(* PLC project Система умного дома.project, CODESYS CODESYS V3.5 SP17 Patch 3 *)
(* stored: creationDateTime 2026-04-06T20:38:17.5908527, modificationDateTime 2026-03-25T09:46:39.3897592 *)

TYPE E_ALERT_PRIORITY : (ALERT_PRIORITY_NONE := 0, ALERT_PRIORITY_LOW := 1, ALERT_PRIORITY_MEDIUM := 2, ALERT_PRIORITY_HIGH := 3, ALERT_PRIORITY_CRITICAL := 4) USINT;
END_TYPE

TYPE E_Behavior_Mode : (BEHAVIOR_HOME := 0, BEHAVIOR_AWAY := 1, BEHAVIOR_NIGHT := 2, BEHAVIOR_MAINTENANCE := 3) INT;
END_TYPE

TYPE E_Gateway_Command_Type : (CMD_NONE := 0, CMD_SET_SCENARIO := 1, CMD_SET_LIGHT := 2, CMD_SET_SOCKET := 3, CMD_SET_SECURITY := 4, CMD_SET_TEMP := 5, CMD_SET_VENT := 6, CMD_SET_BLINDS := 7, CMD_TELEGRAM_MSG := 8, CMD_SYNC_TIME := 9, CMD_RESET_ERRORS := 10, CMD_SET_CONFIG := 11) USINT;
END_TYPE

TYPE E_Lifetime_Device_Type : (LIFETIME_DEVICE_PUMP := 1, LIFETIME_DEVICE_FAN := 2) USINT;
END_TYPE

TYPE E_Outdoor_Mode : (OUTDOOR_MODE_AUTO := 0, OUTDOOR_MODE_PARTY := 1, OUTDOOR_MODE_SECURITY := 2, OUTDOOR_MODE_ECONOMY := 3, OUTDOOR_MODE_MANUAL := 4) USINT;
END_TYPE

TYPE E_PLC_ROLE : (ROLE_UNDEFINED := 0, ROLE_ACTIVE := 1, ROLE_STANDBY := 2, ROLE_OFFLINE := 3) USINT;
END_TYPE

TYPE E_Rule_Action_Type : (ACTION_NONE := 0, ACTION_SET_FLOOR_HEATING := 1, ACTION_SET_LIGHTING_BASE := 2, ACTION_SET_LIGHTING_ACCENT := 3, ACTION_SET_SOCKET := 4, ACTION_SET_VENTILATION := 5, ACTION_SET_BLINDS := 6, ACTION_ACTIVATE_SCENARIO := 7, ACTION_TOGGLE_LIGHTING := 8, ACTION_TOGGLE_SOCKET := 9) USINT;
END_TYPE

TYPE E_Rule_Comparison : (COMP_NONE := 0, COMP_EQ := 1, COMP_GT := 2, COMP_LT := 3, COMP_GE := 4, COMP_LE := 5, COMP_IN_RANGE := 6, COMP_TRUE := 7, COMP_FALSE := 8) USINT;
END_TYPE

TYPE E_Rule_Condition_Type : (COND_NONE := 0, COND_AIR_TEMP := 1, COND_FLOOR_TEMP := 2, COND_HUMIDITY := 3, COND_CO2 := 4, COND_METHANE := 5, COND_CO := 6, COND_DOOR_WINDOW := 7, COND_FLOOD := 8, COND_SMOKE := 9, COND_MOTION := 10, COND_TIME_OF_DAY := 11, COND_DAY_OF_WEEK := 12) USINT;
END_TYPE

TYPE E_SCENARIO_SOURCE : (SRC_NONE := 0, SRC_OPERATOR := 1, SRC_GATEWAY := 2, SRC_RULE := 3, SRC_SAFETY := 4, SRC_POLICY := 5) INT;
END_TYPE

TYPE E_SCENARIO_TYPE : (SCENARIO_NONE := 0, SCENARIO_MORNING := 1, SCENARIO_EVENING := 2, SCENARIO_AWAY := 3, SCENARIO_PARTY := 4, SCENARIO_SLEEP := 5, SCENARIO_EMERGENCY := 6, SCENARIO_PRESENCE := 7) USINT;
END_TYPE

TYPE E_SENSOR_TYPE : (SENSOR_TYPE_NONE := 0, SENSOR_TYPE_DOOR_WINDOW := 5, SENSOR_TYPE_GLASS_BREAK := 6, SENSOR_TYPE_FLOOD := 7, SENSOR_TYPE_SMOKE := 8, SENSOR_TYPE_GAS_METHANE := 1, SENSOR_TYPE_GAS_CO := 2, SENSOR_TYPE_TEMP_FLOOR := 3, SENSOR_TYPE_TEMP_AIR := 4, SENSOR_TYPE_CO2 := 9) USINT;
END_TYPE

TYPE E_System_Operating_Mode : (MODE_NORMAL := 0, MODE_DEGRADED := 1, MODE_SAFE_STOP := 2, MODE_FREEZE_PROTECTION := 3) INT;
END_TYPE

TYPE E_System_Root_Cause : (ROOT_NONE := 0, ROOT_FIRE := 1, ROOT_GAS_LEAK := 2, ROOT_CO_WARNING := 3, ROOT_CO_CRITICAL := 4, ROOT_WATER_LEAK := 5, ROOT_IO_OFFLINE := 6, ROOT_COMM_FAULT := 7, ROOT_SENSOR_FAULT := 8, ROOT_SUBSYSTEM_FAULT := 9, ROOT_WATCHDOG_FAULT := 10) INT;
END_TYPE

TYPE E_System_Severity : (SEV_NORMAL := 0, SEV_WARNING := 1, SEV_DEGRADED := 2, SEV_CRITICAL := 3) INT;
END_TYPE

TYPE E_Trend_Parameter_Type : (TREND_PARAM_NONE := 0, TREND_PARAM_TEMP_AIR := 1, TREND_PARAM_TEMP_FLOOR := 2, TREND_PARAM_PRESSURE := 3, TREND_PARAM_PUMP_CURRENT := 4, TREND_PARAM_GAS_METHANE := 5, TREND_PARAM_GAS_CO := 6) USINT;
END_TYPE

TYPE E_TwoFactor_Method : (TF_METHOD_NONE := 0, TF_METHOD_RFID := 1, TF_METHOD_TOTP := 2, TF_METHOD_BOTH := 3) USINT;
END_TYPE

TYPE E_VALVE_TYPE : (VALVE_NC := 1, VALVE_NO := 2) USINT;
END_TYPE

TYPE E_VENTILATION_LOCATION : (VENT_LOCATION_NONE := 0, VENT_LOCATION_BASEMENT_GAME_ROOM := 1, VENT_LOCATION_BASEMENT_GYM := 2, VENT_LOCATION_BASEMENT_BOILER_ROOM := 3, VENT_LOCATION_BATHROOM_1F := 4, VENT_LOCATION_BATHROOM_2F := 5, VENT_LOCATION_MASTER_BATHROOM := 6, VENT_LOCATION_LAUNDRY := 7, VENT_LOCATION_KITCHEN := 8) USINT;
END_TYPE

TYPE E_VENTILATION_UNIT_TYPE : (VENTILATION_TYPE_NONE := 0, VENTILATION_TYPE_SUPPLY := 1, VENTILATION_TYPE_EXHAUST := 2) USINT;
END_TYPE

TYPE E_Valve_Test_Result : (TEST_RESULT_NONE := 0, TEST_RESULT_PASSED := 1, TEST_RESULT_CURRENT_DEVIATION := 2, TEST_RESULT_TIME_DEVIATION := 3, TEST_RESULT_STALL := 4, TEST_RESULT_LIMIT_SWITCH_FAIL := 5, TEST_RESULT_ABORTED := 6) USINT;
END_TYPE

TYPE E_WEATHER_COMPENSATION_METHOD : (WEATHER_COMP_NONE := 0, WEATHER_COMP_OUTDOOR_RESET := 1) USINT;
END_TYPE

TYPE E_Zone_Access_Level : (ZONE_ACCESS_NONE := 0, ZONE_ACCESS_VIEW := 1, ZONE_ACCESS_CONTROL := 2, ZONE_ACCESS_CONFIG := 3, ZONE_ACCESS_FULL := 4) USINT;
END_TYPE

TYPE ST_Alarm_Record : STRUCT
  ID : UDINT;
  Timestamp_MS : UDINT;
  Source : STRING(20);
  Source_ID : BYTE;
  Message : STRING(100);
  Severity : E_ALERT_PRIORITY;
  Is_Active : BOOL;
  Is_Acknowledged : BOOL;
END_STRUCT;
END_TYPE

TYPE ST_Astro_Time : STRUCT
  sunrise_ms : UDINT := 0;
  sunset_ms : UDINT := 0;
  is_daylight : BOOL := FALSE;
END_STRUCT;
END_TYPE

TYPE ST_BlackBox_Record : STRUCT
  Timestamp : UDINT;
  Gas_Methane_LEL : REAL;
  Gas_CO_PPM : REAL;
  Flood_Active : BOOL;
  Fire_Active : BOOL;
  Valve_Gas_Status : BYTE;
  Valve_Water_Status : BYTE;
  PLC_Active_ID : BYTE;
  System_Mode : BYTE;
  First_Fault_Type : BYTE;
  First_Fault_Source : BYTE;
  First_Fault_Active : BOOL;
  System_Severity : BYTE;
  Root_Cause : BYTE;
  Watchdog_Fault : BOOL;
END_STRUCT;
END_TYPE

TYPE ST_Boiler_Status : STRUCT
  Active : BOOL;
  Running : BOOL;
  Warning : BOOL;
  Error : BOOL;
  Error_ID : WORD;
  Power_Percent : REAL;
  Current_Power : REAL;
  Work_Seconds : UDINT;
  Work_Hours : REAL;
  Resource_Percent : REAL := 100.0;
  Last_Start : DT;
END_STRUCT;
END_TYPE

TYPE ST_Calibration_Family_Summary : STRUCT
  active : BOOL;
  status : INT;
  sensor_count : INT;
  verification_active_count : INT;
  failed_count : INT;
  max_deviation_percent : REAL;
  summary_text : STRING(160);
END_STRUCT;
END_TYPE

TYPE ST_Calibration_Sensor_Summary : STRUCT
  active : BOOL;
  status : INT;
  calibrated_value : REAL;
  deviation_percent : REAL;
  verification_active : BOOL;
  verification_failed : BOOL;
  record_index : INT;
  label : STRING(64);
  summary_text : STRING(160);
END_STRUCT;
END_TYPE

TYPE ST_Component_Maintenance : STRUCT
  Is_Faulty : BOOL;
  Is_In_Maintenance : BOOL;
  Fallback_Value : REAL;
  Use_Last_Good_Value : BOOL;
END_STRUCT;
END_TYPE

TYPE ST_DHW_Config : STRUCT
  Target_Temp : REAL := 55.0;
  Hysteresis : REAL := 2.0;
  Circulation_Schedule_Enabled : BOOL := TRUE;
  Circulation_Start : TOD := TOD#06:00;
  Circulation_End : TOD := TOD#23:00;
  Night_Mode_Enabled : BOOL := TRUE;
  Anti_Legionella_Enabled : BOOL := TRUE;
  Anti_Legionella_Day : UINT := 7;
  Degraded_Target_Delta : REAL := 5.0;
END_STRUCT;
END_TYPE

TYPE ST_DHW_Status : STRUCT
  Temp : REAL;
  Pressure : REAL;
  Heating_Pump_On : BOOL;
  Circ_Pump_On : BOOL;
  Warning : BOOL;
  Error : BOOL;
  Error_ID : WORD;
END_STRUCT;
END_TYPE

TYPE ST_Device_Health : STRUCT
  Health_Score : BYTE := 100;
  Total_Runtime_Hours : UDINT;
  Starts_Count : UDINT;
  Last_Start_Current : REAL;
  Avg_Start_Current : REAL;
  Sample_Count : UDINT;
  Current_Sum : REAL;
  Maintenance_Required : BOOL;
  Warning_Message : STRING(50);
END_STRUCT;
END_TYPE

TYPE ST_Diagnostic_Event : STRUCT
  Code : UDINT;
  Severity : INT;
  Active : BOOL;
  Timestamp : UDINT;
  Source : INT;
END_STRUCT;
END_TYPE

TYPE ST_EVENT : STRUCT
  Event_ID : UDINT;
  Event_Type : UINT;
  Timestamp : UDINT;
  Param1 : UDINT;
  Param2 : UDINT;
END_STRUCT;
END_TYPE

TYPE ST_Flood_Config : STRUCT
  Emergency_Two_Stage_Enabled : BOOL := TRUE;
  Valve_Test_Period_Days : UINT := 7;
  Current_Threshold_MA : REAL := 500.0;
  sensor_to_valve_map : ARRAY[1..GVL_CONSTANTS.C_MAX_FLOOD_SENSORS] OF INT := [1, 1, 1, 1, 2, 2, 2, 2, 3, 3, 3, 3];
END_STRUCT;
END_TYPE

TYPE ST_Flood_Global_Config : STRUCT
  valve_types : ARRAY[1..GVL_CONSTANTS.C_MAX_FLOOD_VALVES] OF E_VALVE_TYPE := [GVL_CONSTANTS.C_MAX_FLOOD_VALVES(E_VALVE_TYPE.VALVE_NC)];
  sensor_to_valve_map : ARRAY[1..GVL_CONSTANTS.C_MAX_FLOOD_SENSORS] OF BYTE := [1, 1, 1, 2, 2, 2, 2, 0, 0, 0];
  min_duration_ms : UDINT := 5000;
  warning_duration_ms : UDINT := 30000;
END_STRUCT;
END_TYPE

TYPE ST_FloorHeating_Circuit_Config : STRUCT
  circuit_id : BYTE := 0;
  zone : BYTE := 0;
  manifold_id : BYTE := 1;
  sensor_id : BYTE := 1;
  valve_id : BYTE := 1;
  control_type : BYTE := 1;
  design_temp : REAL := 35.0;
  min_temp : REAL := 20.0;
  max_temp : REAL := 45.0;
  pid_kp : REAL := 2.0;
  pwm_period_s : UINT := 600;
END_STRUCT;
END_TYPE

TYPE ST_FloorHeating_Global_Config : STRUCT
  enable_floor_heating : BOOL := TRUE;
  anti_freeze_temp : REAL := 7.0;
  overheat_temp : REAL := 45.0;
  weather_compensation_enabled : BOOL := TRUE;
  total_circuits : BYTE := 16;
END_STRUCT;
END_TYPE

TYPE ST_FloorHeating_Manifold_Config : STRUCT
  manifold_id : BYTE;
  location : STRING(30);
  nominal_flow : REAL;
  enable_pump : BOOL;
  circuits : ARRAY[1..GVL_CONSTANTS.C_MAX_CIRCUITS_PER_MANIFOLD] OF ST_FloorHeating_Circuit_Config;
END_STRUCT;
END_TYPE

TYPE ST_Gas_Valve_Configuration : STRUCT
  valve_id : BYTE := 0;
  valve_type : E_VALVE_TYPE := E_VALVE_TYPE.VALVE_NC;
  close_time_seconds : UDINT := 10;
  open_time_seconds : UDINT := 10;
  emergency_open_allowed : BOOL := FALSE;
END_STRUCT;
END_TYPE

TYPE ST_Gateway_Command : STRUCT
  command_id : UDINT;
  timestamp_ms : UDINT;
  operator_id : STRING(10);
  command_type : E_Gateway_Command_Type;
  target_zone : BYTE;
  target_value : REAL;
  target_on_off : BOOL;
  target_scenario : E_SCENARIO_TYPE;
  target_armed : BOOL;
  target_pin : STRING(4);
  target_2fa_code : STRING(6);
  telegram_msg : STRING(200);
  source_ip : STRING(15);
  crc32 : DWORD;
END_STRUCT;
END_TYPE

TYPE ST_Heating_Config : STRUCT
  Weather_Comp_Enabled : BOOL := TRUE;
  Weather_Coef : REAL := 0.1;
  Freeze_Threshold : REAL := 7.0;
  Overheat_Threshold : REAL := 45.0;
  Night_Reduction : REAL := 3.0;
  Target_Floor_Temp : REAL := 28.0;
  Target_Room_Temp : REAL := 22.0;
  Hysteresis : REAL := 0.5;
END_STRUCT;
END_TYPE

TYPE ST_History_Record : STRUCT
  timestamp_ms : UDINT := 0;
  event_code : WORD := 0;
  event_value : REAL := 0.0;
  unit : BYTE := 0;
  zone_id : BYTE := 0;
  operator_id : STRING(10) := '';
  priority : E_ALERT_PRIORITY := E_ALERT_PRIORITY.ALERT_PRIORITY_NONE;
END_STRUCT;
END_TYPE

TYPE ST_Lifetime_Status : STRUCT
  device_id : BYTE;
  runtime_hours : UDINT;
  start_count : UDINT;
  remaining_hours : UDINT;
  remaining_percent : BYTE;
  maintenance_required : BOOL;
  last_calc_timestamp : UDINT;
END_STRUCT;
END_TYPE

TYPE ST_Maintenance_Access_Config : STRUCT
  maintenance_enabled : BOOL := FALSE;
  max_duration_minutes : UDINT := 60;
  requires_two_person : BOOL := TRUE;
  access_level_required : BYTE := 2;
END_STRUCT;
END_TYPE

TYPE ST_Manifold_Status : STRUCT
  Pump_On : BOOL;
  Pump_Current : REAL;
  Pressure : REAL;
  Temp_Supply : REAL;
  Temp_Return : REAL;
  Valve_Pos : REAL;
  Error : BOOL;
  Error_ID : WORD;
  Health : ST_Device_Health;
END_STRUCT;
END_TYPE

TYPE ST_Operator_Zone_Rights : STRUCT
  operator_id : STRING(10);
  global_access_level : BYTE := 0;
  zone_masks : DWORD;
  last_modified : UDINT;
END_STRUCT;
END_TYPE

TYPE ST_Outdoor_Zone_Config : STRUCT
  zone_id : BYTE := 0;
  lighting_circuit_id : BYTE := 0;
  auto_enabled : BOOL := TRUE;
  party_mode_enabled : BOOL := FALSE;
END_STRUCT;
END_TYPE

TYPE ST_Owen_Analog_Value : STRUCT
  rValue : REAL;
  uiCycleTime : UINT;
  wStatus : WORD;
END_STRUCT;
END_TYPE

TYPE ST_Persist : STRUCT
  System_Mode : E_System_Operating_Mode;
  Safety_Gas_Latched : BOOL;
  Safety_Smoke_Latched : BOOL;
  Safety_Leak_Latched : BOOL;
  DHW_Heating_Pump : BOOL;
  Valid : BOOL;
  Version : UINT := 1;
END_STRUCT;
END_TYPE

TYPE ST_Rule : STRUCT
  Action_Type : INT;
  Action_Target_ID : INT;
  Action_Value : REAL;
  Condition_Type : INT;
  Condition_Target_ID : INT;
  Condition_Op : INT;
  Condition_Value : REAL;
  Condition_Value_Max : REAL;
END_STRUCT;
END_TYPE

TYPE ST_Rule_Action : STRUCT
  Active : BOOL;
  Triggered : BOOL;
  Action_Type : E_Rule_Action_Type;
  Target_ID : BYTE;
  Value : REAL;
END_STRUCT;
END_TYPE

TYPE ST_Scenario_Config : STRUCT
  scenario_id : E_SCENARIO_TYPE;
  lighting_level_base : BYTE := 100;
  lighting_level_accent : BYTE := 100;
  floor_heating_adjust_celsius : REAL := 0.0;
  ventilation_speed_percent : BYTE := 50;
  sockets_enabled : BOOL := TRUE;
  blinds_position_percent : BYTE := 0;
  Presence_Simulation_Enabled : BOOL := FALSE;
END_STRUCT;
END_TYPE

TYPE ST_Scenario_Transition_Config : STRUCT
  current_scenario : E_SCENARIO_TYPE;
  target_scenario : E_SCENARIO_TYPE;
  min_duration_minutes : UDINT := 5;
  transition_allowed : BOOL := FALSE;
END_STRUCT;
END_TYPE

TYPE ST_Security_Global_Config : STRUCT
  PIN_Code : STRING(4) := '1234';
  Phones : ARRAY[1..GVL_CONSTANTS.C_MAX_SECURITY_PHONES] OF STRING(15);
  entry_delay_seconds : UDINT := 30;
  exit_delay_seconds : UDINT := 60;
  alarm_duration_seconds : UDINT := 180;
  two_person_timeout_seconds : UDINT := 120;
  max_access_attempts : BYTE := 3;
  auto_arm_enabled : BOOL := FALSE;
  auto_arm_time_ms : UDINT := 0;
  enable_2fa : BOOL := TRUE;
  gate_open_pulse_ms : UDINT := GVL_CONSTANTS.C_MS_IN_SECOND;
  wicket_open_pulse_ms : UDINT := GVL_CONSTANTS.C_MS_IN_SECOND;
  lock_open_pulse_ms : UDINT := GVL_CONSTANTS.C_MS_IN_SECOND;
  lock_close_pulse_ms : UDINT := GVL_CONSTANTS.C_MS_IN_SECOND;
  bypass_motion : ARRAY[1..16] OF BOOL;
  bypass_doors : ARRAY[1..GVL_CONSTANTS.C_MAX_DOOR_SENSORS] OF BOOL;
  bypass_windows : ARRAY[1..16] OF BOOL;
END_STRUCT;
END_TYPE

TYPE ST_Security_Zone_State : STRUCT
  Armed : BOOL;
  Alarm : BOOL;
  Bypassed : BOOL;
  Last_Trigger_Time : DT;
  Trigger_Count : UINT;
END_STRUCT;
END_TYPE

TYPE ST_Sensor_Calibration_Record : STRUCT
  sensor_id : UDINT := 0;
  sensor_type : E_SENSOR_TYPE;
  zone_id : BYTE := 0;
  offset : REAL := 0.0;
  multiplier : REAL := 1.0;
  last_calibration_timestamp : UDINT := 0;
  verification_passed : BOOL := FALSE;
END_STRUCT;
END_TYPE

TYPE ST_State_Snapshot : STRUCT
  timestamp_ms : UDINT := 0;
  operator_id : STRING(10) := '';
  scenario_id : E_SCENARIO_TYPE := E_SCENARIO_TYPE.SCENARIO_NONE;
  lighting_levels : ARRAY[1..GVL_CONSTANTS.C_MAX_LIGHTING_ZONES] OF BYTE;
  floor_heating_setpoints : ARRAY[1..GVL_CONSTANTS.C_MAX_HEATING_CIRCUITS] OF REAL;
  alarm_active : BOOL := FALSE;
  crc32 : DWORD := 0;
END_STRUCT;
END_TYPE

TYPE ST_System_Diagnostics : STRUCT
  Freeze_Hardware_Event_Pending : BOOL;
  Freeze_Hardware_Event_Text : STRING(200);
  Backup_Pump_Fault : BOOL;
  Electric_Heater_Fault : BOOL;
  Backup_Pump_Recovered_After_Retry : BOOL;
  Electric_Heater_Recovered_After_Retry : BOOL;
  Backup_Pump_Out_Of_Service : BOOL;
  Electric_Heater_Out_Of_Service : BOOL;
  Pump_Exercise_Active : BOOL;
  Pump_Exercise_Failed : BOOL;
  Pump_Exercise_Last_Equipment : STRING(80);
  Pump_Exercise_Last_Result : STRING(120);
  Pump_Exercise_No_Feedback_Count : INT;
  Manifold_Pump_Exercise_Count : ARRAY[1..GVL_CONSTANTS.C_MAX_MANIFOLDS] OF UDINT;
  DHW_Heating_Pump_Exercise_Count : UDINT;
  DHW_Circ_Pump_Exercise_Count : UDINT;
  Backup_Pump_Exercise_Count : UDINT;
  Pump_Exercise_Event_Seq : UDINT;
  Pump_Exercise_Journal_1 : STRING(200);
  Pump_Exercise_Journal_2 : STRING(200);
  Pump_Exercise_Journal_3 : STRING(200);
  Pump_Exercise_Journal_Last_Seq : UDINT;
  Pump_Maintenance_Required : BOOL;
  Pump_Maintenance_Warning : BOOL;
  Manifold_Pump_Out_Of_Service : ARRAY[1..GVL_CONSTANTS.C_MAX_MANIFOLDS] OF BOOL;
  DHW_Heating_Pump_Out_Of_Service : BOOL;
  DHW_Circ_Pump_Out_Of_Service : BOOL;
  Maintenance_Last_Action : STRING(120);
  Operator_Action_Blocked : BOOL;
  Operator_Block_Reason : STRING(160);
  Operator_Last_Forbidden_Action : STRING(160);
  Operator_Journal_1 : STRING(200);
  Operator_Journal_2 : STRING(200);
  Operator_Journal_3 : STRING(200);
  Operator_Journal_Event_Seq : UDINT;
  Operator_Journal_Last_Seq : UDINT;
  Dangerous_Action_Pending_Confirm : BOOL;
  Dangerous_Action_Confirm_Text : STRING(160);
  Dangerous_Action_Confirm_Deadline_MS : UDINT;
  User_Access_Level_Active : INT;
  User_Access_Denied : BOOL;
  User_Access_Deny_Reason : STRING(160);
  Valve_Test_Mode_Active : BOOL;
  Valve_Test_Deadline_MS : UDINT;
  Valve_Test_Remaining_MS : UDINT;
  Valve_Test_Validation_OK : BOOL;
  Valve_Test_Validation_Text : STRING(160);
  Valve_Test_Forced_Close : BOOL;
  Water_Valve_Test_Mode_Active : BOOL;
  Water_Valve_Test_Deadline_MS : UDINT;
  Water_Valve_Test_Remaining_MS : UDINT;
  Water_Valve_Test_Validation_OK : BOOL;
  Water_Valve_Test_Validation_Text : STRING(160);
  Water_Valve_Test_Forced_Close : BOOL;
  Gas_Valve_Test_Mode_Active : BOOL;
  Gas_Valve_Test_Deadline_MS : UDINT;
  Gas_Valve_Test_Remaining_MS : UDINT;
  Gas_Valve_Test_Validation_OK : BOOL;
  Gas_Valve_Test_Validation_Text : STRING(160);
  Gas_Valve_Test_Forced_Close : BOOL;
  Active_Leak_Sensor_Index : INT;
  Active_Gas_Sensor_Index : INT;
  Active_Leak_Zone_Name : STRING(80);
  Active_Gas_Zone_Name : STRING(80);
  Water_Valve_Test_Context : STRING(160);
  Gas_Valve_Test_Context : STRING(160);
  Water_Recovery_Target_Zone_Index : INT;
  Gas_Recovery_Target_Zone_Index : INT;
  Water_Recovery_Selective_Allowed : BOOL;
  Gas_Recovery_Selective_Allowed : BOOL;
  Water_Recovery_Selective_Text : STRING(160);
  Gas_Recovery_Selective_Text : STRING(160);
  Water_Recovery_Physical_Active : BOOL;
  Water_Recovery_Physical_Zone_Name : STRING(80);
  Water_Zone_Open_Fault : ARRAY[1..32] OF BOOL;
  Water_Zone_Close_Fault : ARRAY[1..32] OF BOOL;
  Water_Valve_Exercise_Last_Zone : INT;
  Water_Valve_Exercise_Last_Result : STRING(160);
  Water_Zone_Critical_Close_Fault : ARRAY[1..32] OF BOOL;
  Water_Close_Fault_Active : BOOL;
  Water_Close_Fault_Zone_Name : STRING(80);
  Water_Close_Fault_Text : STRING(200);
  Water_Zone_Close_Retry_Active : ARRAY[1..32] OF BOOL;
  Water_Zone_Close_Retry_Count : ARRAY[1..32] OF INT;
  Water_Zone_Close_Recovered_After_Retry : ARRAY[1..32] OF BOOL;
  Water_Localization_Failed : BOOL;
  Water_Main_Shutdown_Recommended : BOOL;
  Water_Escalation_Text : STRING(200);
  Alarm_Event_Pulse : BOOL;
  Alarm_Event_Code : UDINT;
  Alarm_Event_Value : REAL;
  Sensor_Fault : BOOL;
  IO_Offline : BOOL;
  Subsystem_Degraded : BOOL;
  Manifold_Pressure_Fault : ARRAY[1..GVL_CONSTANTS.C_MAX_MANIFOLDS] OF BOOL;
  Manifold_Pressure_Diag_Code : ARRAY[1..GVL_CONSTANTS.C_MAX_MANIFOLDS] OF WORD;
  Manifold_Pressure_Fault_Active : BOOL;
  Manifold_Pressure_First_Fault_Index : INT;
  Manifold_Pressure_Fault_Text : STRING(160);
  Manifold_Current_Fault : ARRAY[1..GVL_CONSTANTS.C_MAX_MANIFOLDS] OF BOOL;
  Manifold_Current_Diag_Code : ARRAY[1..GVL_CONSTANTS.C_MAX_MANIFOLDS] OF WORD;
  Manifold_Current_Fault_Active : BOOL;
  Manifold_Current_First_Fault_Index : INT;
  Manifold_Current_Fault_Text : STRING(160);
  Manifold_Return_Temp_Fault : ARRAY[1..GVL_CONSTANTS.C_MAX_MANIFOLDS] OF BOOL;
  Manifold_Return_Temp_Diag_Code : ARRAY[1..GVL_CONSTANTS.C_MAX_MANIFOLDS] OF WORD;
  Manifold_Return_Temp_Fault_Active : BOOL;
  Manifold_Return_Temp_First_Fault_Index : INT;
  Manifold_Return_Temp_Fault_Text : STRING(160);
  Manifold_Sensor_Fault_Count : ARRAY[1..GVL_CONSTANTS.C_MAX_MANIFOLDS] OF INT;
  Manifold_Sensor_Out_Of_Service : ARRAY[1..GVL_CONSTANTS.C_MAX_MANIFOLDS] OF BOOL;
  Manifold_Sensor_Out_Of_Service_Active : BOOL;
  Manifold_Sensor_First_OOS_Index : INT;
  Manifold_Sensor_OOS_Text : STRING(160);
END_STRUCT;
END_TYPE

TYPE ST_System_State_Snapshot : STRUCT
  System_Time_MS : UDINT;
  Current_Scenario : E_SCENARIO_TYPE;
  Security_Armed : BOOL;
  Active_Alarms : INT;
  Zone_Valves : ARRAY[1..GVL_CONSTANTS.C_MAX_HEATING_CIRCUITS] OF BOOL;
  Manifold_Pumps : ARRAY[1..GVL_CONSTANTS.C_MAX_MANIFOLDS] OF BOOL;
  Lighting_States : ARRAY[1..32] OF BYTE;
  Blinds_Positions : ARRAY[1..GVL_CONSTANTS.C_MAX_BLINDS] OF BYTE;
  Socket_States : ARRAY[1..GVL_CONSTANTS.C_MAX_SOCKETS] OF BOOL;
  Gas_Valve_Closed : BOOL;
  Water_Valves_Closed : BOOL;
  Version : UDINT;
END_STRUCT;
END_TYPE

TYPE ST_System_State_Summary : STRUCT
  Outdoor_Temp : REAL;
  Indoor_Temp : ARRAY[1..GVL_CONSTANTS.C_MAX_CLIMATE_ZONES] OF REAL;
  Floor_Temps : ARRAY[1..GVL_CONSTANTS.C_MAX_HEATING_CIRCUITS] OF REAL;
  Humidity : ARRAY[1..GVL_CONSTANTS.C_MAX_HUMIDITY_SENSORS] OF REAL;
  CO2 : ARRAY[1..GVL_CONSTANTS.C_MAX_CO2_SENSORS] OF REAL;
  Gas_Alarm : BOOL;
  Flood_Alarm : BOOL;
  Fire_Alarm : BOOL;
  Security_Alarm : BOOL;
  Security_Armed : BOOL;
END_STRUCT;
END_TYPE

TYPE ST_Tariff_Config : STRUCT
  Enabled : BOOL := FALSE;
  Night_Start_Hour : UINT := 23;
  Night_End_Hour : UINT := 7;
  Boost_Delta : REAL := 2.0;
END_STRUCT;
END_TYPE

TYPE ST_Trend_Config : STRUCT
  param_type : BYTE;
  zone_id : BYTE;
  enabled : BOOL;
  deviation_threshold_percent : REAL := 10.0;
  history_days : UDINT := 7;
END_STRUCT;
END_TYPE

TYPE ST_Trend_Data : STRUCT
  config : ST_Trend_Config;
  record_count : UDINT;
  write_index : UDINT;
  sum_values : REAL;
  values : ARRAY[1..100] OF REAL;
  timestamps : ARRAY[1..100] OF UDINT;
  crc32 : DWORD;
END_STRUCT;
END_TYPE

TYPE ST_Trend_Header : STRUCT
  parameter_type : BYTE;
  zone_id : BYTE := 0;
  records_count : UDINT := 0;
  average_value : REAL := 0.0;
  min_value : REAL := 0.0;
  max_value : REAL := 0.0;
END_STRUCT;
END_TYPE

TYPE ST_Trend_History_Record : STRUCT
  timestamp_ms : UDINT := 0;
  value : REAL := 0.0;
END_STRUCT;
END_TYPE

TYPE ST_TwoFactor_Auth_State : STRUCT
  Auth_Method : E_TwoFactor_Method;
  is_pending : BOOL;
  Attempts_Left : UINT;
  Time_Left_S : UINT;
  Is_Success : BOOL;
  Is_Locked : BOOL;
END_STRUCT;
END_TYPE

TYPE ST_TwoFactor_Data : STRUCT
  operator_id : STRING(10);
  AuthMethod : BYTE;
  rfid_tag : STRING(20);
  totp_secret : STRING(32);
  last_modified : UDINT;
END_STRUCT;
END_TYPE

TYPE ST_User_Rule : STRUCT
  Enabled : BOOL;
  Condition_Type : E_Rule_Condition_Type;
  Condition_Target_ID : BYTE;
  Condition_Op : E_Rule_Comparison;
  Condition_Value : REAL;
  Condition_Value_Max : REAL;
  Action_Target_ID : BYTE;
  Action_Value : REAL;
  Action_Type : E_Rule_Action_Type;
  Priority : BYTE;
END_STRUCT;
END_TYPE

TYPE ST_Valve_Test_Config : STRUCT
  valve_id : BYTE := 0;
  test_interval_days : UDINT := 7;
  Nominal_Current : REAL := 0.5;
  nominal_close_time_sec : REAL := 10.0;
  enabled : BOOL := TRUE;
END_STRUCT;
END_TYPE

TYPE ST_Ventilation_Config : STRUCT
  CO2_Threshold : REAL := 800.0;
  Humidity_Threshold : REAL := 65.0;
  Night_Mode_Start : TOD := TOD#23:00;
  Night_Mode_End : TOD := TOD#07:00;
END_STRUCT;
END_TYPE

TYPE ST_Ventilation_Global_Config : STRUCT
  enable_ventilation : BOOL := TRUE;
  total_units : BYTE := 8;
  default_supply_speed : BYTE := 40;
  default_exhaust_speed : BYTE := 40;
  Degraded_Exhaust_Limit : BYTE := 30;
  Scenario_Modes : ARRAY[1..GVL_CONSTANTS.C_MAX_SCENARIOS] OF ST_Ventilation_Scenario_Mode;
  wet_zone_to_exhaust_map : ARRAY[1..GVL_CONSTANTS.C_MAX_WET_ZONES] OF INT := [2, 3, 4, 5];
  pv3_exhaust_index : INT := 3;
END_STRUCT;
END_TYPE

TYPE ST_Ventilation_Scenario_Mode : STRUCT
  Scenario_ID : BYTE;
  Scenario_Priority : BYTE;
  Fire_Alarm : BOOL;
  Methane_Alarm : BOOL;
  Smoke_Detected : BOOL;
  Exhaust_Modes : ARRAY[1..GVL_CONSTANTS.C_MAX_EXHAUST_FANS] OF BYTE;
  Supply_Modes : ARRAY[1..GVL_CONSTANTS.C_MAX_SUPPLY_FANS] OF BYTE;
  Base_Fan_Speed : BYTE := 50;
  Target_Temp : REAL := 22.0;
END_STRUCT;
END_TYPE

TYPE ST_Ventilation_Unit : STRUCT
  Enabled : BOOL;
  Speed_Percent : REAL;
  Filter_Dirty : BOOL;
  Error : BOOL;
  Mode : BYTE;
END_STRUCT;
END_TYPE

TYPE ST_Ventilation_Unit_Config : STRUCT
  unit_id : BYTE := 0;
  unit_type : E_VENTILATION_UNIT_TYPE;
  location : E_VENTILATION_LOCATION;
  min_speed : BYTE := 20;
  max_speed : BYTE := 100;
  Threshold_Hum : REAL := 65.0;
  has_smoke_detector : BOOL := FALSE;
END_STRUCT;
END_TYPE

TYPE ST_Zone_Sensors : STRUCT
  Temp_Room : REAL;
  Temp_Floor : REAL;
  Motion_Active : BOOL;
  Switch_Physical : BOOL;
  Light_State : BOOL;
  Maintenance : ST_Component_Maintenance;
END_STRUCT;
END_TYPE

{attribute 'qualified_only'}
VAR_GLOBAL  (* GVL_TEST_PANEL *)
  G_Enable : BOOL := FALSE;
  G_Scenario_ID : INT := 1;
  G_Scenario_ID_Prev : INT := 0;
  G_Scenario_Run : BOOL := FALSE;
  G_Scenario_Active : BOOL := FALSE;
  G_UI_00_Header : STRING(200) := '=== TEST PANEL ===';
  G_UI_01_Test : STRING(200) := 'Select G_Scenario_ID';
  G_UI_02_Change : STRING(200) := 'CHANGE: set scenario inputs';
  G_UI_03_Expected : STRING(200) := 'EXPECTED: see scenario instruction';
  G_UI_04_Result : STRING(200) := 'RESULT: Idle';
  G_UI_05_Error : STRING(200) := 'ERROR: -';
  G_UI_06_Actual : STRING(200) := 'ACTUAL: see numeric fields below';
  G_UI_07_Separator : STRING(200) := '----------------------------------------';
  G_UI_10_Numeric_Block : STRING(200) := 'NUMERIC: Base / Expected / Actual / Delta';
  G_UI_11_Array_Block : STRING(200) := 'ARRAYS: Manifold expected / actual / enabled';
  G_UI_12_State_Block : STRING(200) := 'STATE: Safety / Block / Budget / Preheat';
  G_Run_Counter : UDINT := 0;
  G_Last_Scenario_ID : INT := 0;
  G_Last_Result_Passed : BOOL := TRUE;
  G_Last_Fail_Code : UDINT := 0;
  G_Reset_Results_Request : BOOL := FALSE;
  G_Reset_Inputs_Request : BOOL := FALSE;
  G_Current_Test_Name : STRING(200) := '';
  G_Expected_Summary : STRING(200) := '';
  G_Actual_Summary : STRING(200) := '';
  G_Test_Result_Line : STRING(200) := 'Idle';
  G_Last_Result_Line : STRING(200) := '';
  G_Error_Text : STRING(200) := '';
  G_System_State_Line : STRING(200) := '';
  G_Selected_Circuit : INT := 1;
  G_Input_Policy_Bias : INT := 0;
  G_Input_Guest_Preheat_Request : BOOL := FALSE;
  G_Input_Guest_Preheat_Enabled : BOOL := TRUE;
  G_Input_Guest_Preheat_Boost : INT := 2;
  G_Input_Max_Thermal_Budget : REAL := 2.0;
  G_Input_Block_Heating : BOOL := FALSE;
  G_Input_Safety_Stop : BOOL := FALSE;
  G_Input_Circuit_Enable : ARRAY[1..GVL_CONSTANTS.C_MAX_HEATING_CIRCUITS] OF BOOL;
  G_Input_Circuit_Bias : ARRAY[1..GVL_CONSTANTS.C_MAX_HEATING_CIRCUITS] OF INT;
  G_Input_Circuit_Guest_Preheat : ARRAY[1..GVL_CONSTANTS.C_MAX_HEATING_CIRCUITS] OF BOOL;
  G_Test_Description : STRING(200) := 'Idle';
  G_Test_What_To_Change : STRING(200) := '';
  G_Test_Expected_Text : STRING(200) := '';
  G_Result_Mapped_Manifold : INT := 0;
  G_Result_Base_Priority : INT := 0;
  G_Result_Expected_Adjusted_Priority : INT := 0;
  G_Result_Actual_Adjusted_Priority : INT := 0;
  G_Result_Delta : INT := 0;
  G_Result_Manifold_Base_Priority : ARRAY[1..GVL_CONSTANTS.C_MAX_MANIFOLDS] OF INT;
  G_Result_Manifold_Expected_Priority : ARRAY[1..GVL_CONSTANTS.C_MAX_MANIFOLDS] OF INT;
  G_Result_Manifold_Actual_Priority : ARRAY[1..GVL_CONSTANTS.C_MAX_MANIFOLDS] OF INT;
  G_Result_Manifold_Delta : ARRAY[1..GVL_CONSTANTS.C_MAX_MANIFOLDS] OF INT;
  G_Result_Manifold_Allowed : ARRAY[1..GVL_CONSTANTS.C_MAX_MANIFOLDS] OF BOOL;
  G_Result_Manifold_Enabled : ARRAY[1..GVL_CONSTANTS.C_MAX_MANIFOLDS] OF BOOL;
  G_Result_Used_Thermal_Budget : REAL := 0.0;
  G_Result_Budget_Exceeded : BOOL := FALSE;
  G_Result_Passed : BOOL := TRUE;
  G_Result_Status_Msg : STRING(200) := 'Idle';
  G_Result_Fail_Code : UDINT := 0;
END_VAR

VAR_GLOBAL  (* GVL_COMMAND_VERIFY *)
  Command_Mismatch_Count : INT := 0;
  Command_Match_OK : BOOL := TRUE;
  Command_Mismatch_Active : BOOL := FALSE;
END_VAR

VAR_GLOBAL  (* GVL_POLICY *)
  G_Rule_Preheat_Request : BOOL := FALSE;
  G_Scenario_Request_Operator : E_SCENARIO_TYPE := E_SCENARIO_TYPE.SCENARIO_NONE;
  G_Scenario_Request_Gateway : E_SCENARIO_TYPE := E_SCENARIO_TYPE.SCENARIO_NONE;
  G_Scenario_Request_Rule : E_SCENARIO_TYPE := E_SCENARIO_TYPE.SCENARIO_NONE;
  G_Scenario_Intent : E_SCENARIO_TYPE := E_SCENARIO_TYPE.SCENARIO_NONE;
  G_Scenario_Source : E_SCENARIO_SOURCE := SRC_NONE;
END_VAR

{attribute 'qualified_only'}
VAR_GLOBAL  (* GVL_TEST_PANEL_RESULT *)
  G_Enable : BOOL := FALSE;
  G_Scenario_ID : INT := 0;
  G_Scenario_Run : BOOL := FALSE;
  G_Scenario_Active : BOOL := FALSE;
  G_Test_Result_Line : STRING(200) := 'Idle';
  G_Result_Passed : BOOL := FALSE;
  G_Result_Status_Msg : STRING(200) := 'Idle';
  G_Result_Fail_Code : UDINT := 0;
  G_Result_Base_Priority : INT := 0;
  G_Result_Expected_Adjusted_Priority : INT := 0;
  G_Result_Actual_Adjusted_Priority : INT := 0;
  G_Result_Delta : INT := 0;
  G_Result_Budget_Exceeded : BOOL := FALSE;
  G_Result_Used_Thermal_Budget : REAL := 0.0;
  G_Result_Manifold_Enabled : ARRAY[1..GVL_CONSTANTS.C_MAX_MANIFOLDS] OF BOOL;
END_VAR

VAR_GLOBAL  (* GVL_HEATING_REQUEST *)
  G_Freeze_Request : BOOL := FALSE;
  G_Target_Temperature : REAL := 0.0;
  G_Preheat_Request : BOOL := FALSE;
END_VAR

VAR_GLOBAL  (* GVL_INTENT_SYSTEM *)
  I_Source_Valid : BOOL := FALSE;
  I_Last_Update_Cycle : UDINT := 0;
  I_Last_Update_MS : UDINT := 0;
  I_Mode_Safe_Stop_Active : BOOL := FALSE;
  I_Mode_Degraded_Active : BOOL := FALSE;
  I_Mode_Freeze_Protection_Active : BOOL := FALSE;
  I_Preheat_Request : BOOL := FALSE;
  I_Freeze_Request : BOOL := FALSE;
  I_Scenario_Request_Allowed : BOOL := FALSE;
  I_Operator_Scenario_Block : BOOL := FALSE;
  I_Gateway_Command_Valid : BOOL := FALSE;
  I_Gateway_Command_Type : INT := 0;
  I_Gateway_Writes_Allowed : BOOL := FALSE;
  I_Reset_Errors_Request : BOOL := FALSE;
  I_Config_Apply_Allowed : BOOL := FALSE;
  I_Time_Sync_Allowed : BOOL := FALSE;
  I_Temperature_Write_Allowed : BOOL := FALSE;
  I_Ventilation_Write_Allowed : BOOL := FALSE;
  I_Maintenance_Apply_Allowed : BOOL := FALSE;
  I_Lighting_Overrides_Block : BOOL := FALSE;
  I_Blinds_Overrides_Block : BOOL := FALSE;
  I_Socket_Overrides_Block : BOOL := FALSE;
  I_Access_Open_Allowed : BOOL := FALSE;
  I_Manual_Override_Allowed : BOOL := FALSE;
  I_Dangerous_Action_Allowed : BOOL := FALSE;
END_VAR

{attribute 'qualified_only'}
VAR_GLOBAL CONSTANT  (* GVL_CONSTANTS *)
  C_MAX_ZONES : INT := 16;  (* Максимальное количество зон (комнат) *)
  C_MAX_LIGHTING_ZONES : INT := 32;  (* Алиас для контуров освещения *)
  C_MAX_HEATING_CIRCUITS : INT := 16;  (* Количество физических контуров теплого пола по ТЗ *)
  C_MAX_CLIMATE_ZONES : INT := 16;  (* Алиас для климатических зон *)
  C_MAX_LIGHT_ZONES : INT := 32;  (* Алиас для световых зон *)
  C_MAX_SOCKETS : INT := 36;  (* Максимальное количество управляемых розеток *)
  C_MAX_BLINDS : INT := 20;  (* Максимальное количество штор/жалюзи *)
  C_MAX_ALARMS : INT := 20;  (* Максимальное количество активных тревог *)
  C_MAX_RULES : INT := 20;  (* Максимальное количество правил (движок правил) *)
  C_MAX_MANIFOLDS : INT := 5;  (* Максимальное количество коллекторов *)
  C_MAX_BOILERS : INT := 2;  (* Максимальное количество котлов *)
  C_MAX_SUPPLY_FANS : INT := 3;  (* Максимальное количество приточных вентиляторов *)
  C_MAX_EXHAUST_FANS : INT := 5;  (* Максимальное количество вытяжных вентиляторов *)
  C_MAX_SECURITY_SENSORS : INT := 15;  (* Максимальное количество датчиков безопасности (герконы, стекло) *)
  C_MAX_FLOOD_SENSORS : INT := 12;  (* Максимальное количество датчиков протечки *)
  C_MAX_DOOR_SENSORS : INT := 8;  (* Максимальное количество датчиков дверей *)
  C_MAX_CO_SENSORS : INT := 8;  (* Максимальное количество датчиков CO *)
  C_MAX_METHANE_SENSORS : INT := 2;  (* Максимальное количество датчиков метана *)
  C_MAX_VENT_UNITS : INT := 8;  (* Максимальное количество вентустановок *)
  C_MAX_SUPPLY_TEMPS : INT := 2;  (* Максимальное количество датчиков температуры притока *)
  C_MAX_SMOKE_SENSORS : INT := 6;  (* Максимальное количество датчиков дыма *)
  C_MAX_SCENARIOS : INT := 6;  (* Максимальное количество сценариев *)
  C_MAX_OUTDOOR_ZONES : INT := 4;  (* Максимальное количество зон уличного освещения *)
  C_MAX_ACCESS_CODES : INT := 10;  (* Максимальное количество кодов доступа *)
  C_MAX_WET_ZONES : INT := 4;  (* Максимальное количество "мокрых" зон (санузлы) *)
  C_MAX_CALIBRATIONS : INT := 20;  (* Максимальное количество калибровок датчиков *)
  C_MAX_MODULES : INT := 10;  (* Максимальное количество модулей ввода-вывода *)
  C_MAX_CLEANING_MODES : INT := 3;  (* Максимальное количество режимов уборки *)
  C_MAX_ALLOWED_IPS : INT := 5;  (* Максимальное количество разрешенных IP-адресов *)
  C_MAX_VENT_SUPPLY_MODES : INT := 3;  (* Максимальное количество режимов притока вентиляции *)
  C_MAX_SECURITY_PHONES : INT := 5;  (* Максимальное количество телефонов для оповещения *)
  C_MAX_FLOOD_VALVES : INT := 3;  (* Максимальное количество кранов защиты от протечек *)
  C_MAX_HUMIDITY_SENSORS : INT := 8;  (* Максимальное количество датчиков влажности *)
  C_MAX_CO2_SENSORS : INT := 8;  (* Максимальное количество датчиков CO2 *)
  C_MAX_CIRCUITS_PER_MANIFOLD : INT := 4;  (* Максимальное количество контуров на коллектор *)
  C_MAX_TREND_DATA_POINTS : INT := 100;  (* Максимальное количество точек данных для трендов *)
  C_MAX_HISTORY_RECORDS : INT := 100;  (* Максимальное количество записей в истории *)
  C_MAX_DEBUG_LOGS : INT := 1000;  (* Максимальное количество записей в логе отладки *)
  C_MAX_GATEWAY_COMMANDS : INT := 10;  (* Максимальное количество команд в буфере шлюза *)
  C_MAX_STATE_SNAPSHOTS : INT := 10;  (* Максимальное количество снимков состояния *)
  C_MAX_BLACKBOX_RECORDS : INT := 100;  (* Максимальное количество записей черного ящика *)
  C_MAX_PRESENCE_HISTORY : INT := 1008;  (* Максимальное количество записей истории присутствия *)
  C_MAX_MODBUS_REGISTERS : INT := 201;  (* Максимальное количество регистров Modbus *)
  C_MAX_DEDUPLICATION_HISTORY : INT := 100;  (* Максимальное количество записей истории дедупликации *)
  C_MAX_NVRAM_RECORDS : INT := 100;  (* Максимальное количество записей NVRAM *)
  C_MAX_NVRAM_DATA : INT := 128;  (* Максимальный размер данных NVRAM *)
  C_ANALOG_RAW_MAX : WORD := 27648;  (* Максимальное значение АЦП (100%) *)
  C_ANALOG_4MA_RAW : WORD := 5529;  (* Значение АЦП для 4mA (20% от 27648) *)
  C_ANALOG_3_6MA_RAW : WORD := 4976;  (* Порог обрыва NAMUR NE43 (< 3.6mA) *)
  C_ANALOG_21MA_RAW : WORD := 29030;  (* Порог КЗ NAMUR NE43 (> 21mA) *)
  C_ANALOG_10V_MAX_RAW : WORD := 30000;  (* Порог выхода за пределы 0-10V *)
  C_MS_IN_SECOND : UDINT := 1000;
  C_MS_IN_MINUTE : UDINT := 60000;
  C_MS_IN_HOUR : UDINT := 3600000;
  C_MS_IN_DAY : UDINT := 86400000;
  C_BOILER_CASCADE_MIN_DEMAND : REAL := 25.0;  (* Минимальный запрос для включения ведущего котла (5% от одного коллектора) *)
  C_BOILER_CASCADE_HIGH_DEMAND : REAL := 250.0;  (* Высокий запрос для включения второго котла (50% от общей мощности) *)
END_VAR

VAR_GLOBAL  (* GVL_INTENT_SAFETY *)
  I_Source_Valid : BOOL := FALSE;
  I_Last_Update_Cycle : UDINT := 0;
  I_Last_Update_MS : UDINT := 0;
  I_Fire_Alarm_Active : BOOL := FALSE;
  I_Gas_Alarm_Active : BOOL := FALSE;
  I_Leak_Alarm_Active : BOOL := FALSE;
  I_CO_Warning_Active : BOOL := FALSE;
  I_System_Safe_Stop_Required : BOOL := FALSE;
  I_Freeze_Protection_Required : BOOL := FALSE;
  I_Evacuation_Mode_Active : BOOL := FALSE;
  I_Gas_Close_Required : BOOL := FALSE;
  I_Boiler_Stop_Required : BOOL := FALSE;
  I_Vent_Stop_Required : BOOL := FALSE;
  I_Vent_Force_PV3_Boost : BOOL := FALSE;
  I_Vent_Force_Supply_100 : BOOL := FALSE;
  I_Vent_Force_Supply_80 : BOOL := FALSE;
  I_Vent_Force_Exhaust_100 : BOOL := FALSE;
  I_Water_Main_Close_Required : BOOL := FALSE;
  I_Water_Zone_Close_Required : ARRAY[1..32] OF BOOL;
  I_Water_Selective_Recovery_Allowed : BOOL := FALSE;
  I_Water_Recovery_Target_Zone : INT := 0;
  I_Lock_1_Force_Open : BOOL := FALSE;
  I_Lock_1_Force_Close_Block : BOOL := FALSE;
  I_Lock_2_Force_Open : BOOL := FALSE;
  I_Lock_2_Force_Close_Block : BOOL := FALSE;
END_VAR

{attribute 'qualified_only'}
VAR_GLOBAL  (* GVL_COMMAND *)
  G_Gas_Valve_Close : BOOL := FALSE;  (* Команда: Закрыть газовый клапан *)
  G_Boiler_Stop : BOOL := FALSE;  (* Команда: Остановка котлов *)
  G_Supply_100_Req : BOOL := FALSE;  (* Команда: Приток 100% *)
  G_Supply_80_Req : BOOL := FALSE;  (* Команда: Приток 80% *)
  G_Vent_PV3_Boost : BOOL := FALSE;  (* Команда: Форсированный режим ПВ-3 *)
  G_Exhaust_100_Req : BOOL := FALSE;  (* Команда: Вытяжка 100% *)
  G_Vent_Stop : BOOL := FALSE;  (* Команда: Остановка вентиляции *)
  G_Close_Valve_35 : BOOL := FALSE;  (* Команда: Закрыть вводной кран 1 *)
  G_Close_Valve_36 : BOOL := FALSE;  (* Команда: Закрыть вводной кран 2 *)
  G_Gate_Open : BOOL;
  G_Wicket_Open : BOOL;
  G_Lock_1_Open : BOOL;
  G_Lock_1_Close : BOOL;
  G_Lock_2_Open : BOOL;
  G_Lock_2_Close : BOOL;
  G_Reset_Errors : BOOL := FALSE;  (* Команда: Сброс ошибок *)
  G_Scenario_Request : E_SCENARIO_TYPE := E_SCENARIO_TYPE.SCENARIO_NONE;
  G_Scenario_Request_Operator : E_SCENARIO_TYPE := E_SCENARIO_TYPE.SCENARIO_NONE;  (* Запрос на активацию сценария *)
  G_Arm_Req : BOOL;
  G_Disarm_Req : BOOL;
  G_PIN_Code : STRING(4);
  G_RFID_Tag : STRING(20);
  G_2FA_Code_In : STRING(6);
  G_Send_2FA_Req : BOOL;
  G_2FA_Code_Out : STRING(6);
  G_Lighting_Override : ARRAY[1..32] OF BYTE;
  G_Blinds_Override : ARRAY[1..GVL_CONSTANTS.C_MAX_BLINDS] OF BYTE;
  G_Socket_Override : ARRAY[1..GVL_CONSTANTS.C_MAX_SOCKETS] OF BOOL;
  CMD_Set_Manifold_Pump_In_Service : ARRAY[1..GVL_CONSTANTS.C_MAX_MANIFOLDS] OF BOOL;
  CMD_Set_DHW_Heating_Pump_In_Service : BOOL;
  CMD_Set_DHW_Circ_Pump_In_Service : BOOL;
  CMD_Dangerous_Action_Confirm : BOOL;
  CMD_Dangerous_Action_Request : BOOL;
  CMD_User_Access_Level : INT := 0;
  CMD_Valve_Test_Open : BOOL;
  CMD_Valve_Test_Close : BOOL;
  CMD_Valve_Test_Confirm : BOOL;
  CMD_Water_Valve_Test_Open : BOOL;
  CMD_Water_Valve_Test_Close : BOOL;
  CMD_Water_Valve_Test_Confirm : BOOL;
  CMD_Gas_Valve_Test_Open : BOOL;
  CMD_Gas_Valve_Test_Close : BOOL;
  CMD_Gas_Valve_Test_Confirm : BOOL;
  CMD_Water_Selective_Recover : BOOL;
  CMD_Gas_Selective_Recover : BOOL;
END_VAR

{attribute 'qualified_only'}
VAR_GLOBAL  (* GVL_SYSTEM_COORDINATION *)
  G_System_Degraded : BOOL := FALSE;
  G_Block_Heating : BOOL := FALSE;
  G_Block_Ventilation : BOOL := FALSE;
  G_Block_Lighting_Override : BOOL := FALSE;
  G_Block_Sockets_Override : BOOL := FALSE;
  G_Coordination_Code : UDINT := 0;
  G_Coordination_Status_Msg : STRING(200) := '';
END_VAR

{attribute 'qualified_only'}
VAR_GLOBAL  (* GVL_IO *)
  DI_Security_Open : ARRAY[1..GVL_CONSTANTS.C_MAX_SECURITY_SENSORS] OF BOOL;  (* Дискретные входы: Герконы (нормально-замкнутые контакты, TRUE = Открыто) *)
  DI_Security_Glass : ARRAY[1..GVL_CONSTANTS.C_MAX_SECURITY_SENSORS] OF BOOL;  (* Дискретные входы: Датчики разбития стекла (активный уровень - TRUE) *)
  DI_Security_2F_Group : BOOL;  (* Дискретный вход: Групповой шлейф безопасности 2-го этажа (общий сигнал) *)
  DI_Flood_Sensors : ARRAY[1..GVL_CONSTANTS.C_MAX_FLOOD_SENSORS] OF BOOL;  (* Дискретные входы: Датчики протечки воды (активный уровень - TRUE) *)
  DI_Manifold_End_Switches : ARRAY[1..GVL_CONSTANTS.C_MAX_MANIFOLDS] OF BOOL;  (* Дискретные входы: Концевые выключатели клапанов коллекторов *)
  AO_Manifold_Valves : ARRAY[1..GVL_CONSTANTS.C_MAX_MANIFOLDS] OF UINT;  (* Аналоговые выходы: Приводы клапанов (0-10В, 0-1000 ед. для Modbus) *)
  DO_Manifold_Pumps : ARRAY[1..GVL_CONSTANTS.C_MAX_MANIFOLDS] OF BOOL;  (* Дискретные выходы: Циркуляционные насосы коллекторных узлов (220В) *)
  AI_Manifold_Currents : ARRAY[1..GVL_CONSTANTS.C_MAX_MANIFOLDS] OF INT;  (* Аналоговые входы: Обратная связь по току потребления насосов (диагностика) *)
  AI_Manifold_Pressures : ARRAY[1..GVL_CONSTANTS.C_MAX_MANIFOLDS] OF INT;  (* Аналоговые входы: Давление теплоносителя в коллекторах (0-10 бар) *)
  AI_Manifold_Temps_Supply : ARRAY[1..GVL_CONSTANTS.C_MAX_MANIFOLDS] OF ST_Owen_Analog_Value;  (* Аналоговые входы: Температура подачи (структура со статусом) *)
  AI_Manifold_Temps_Return : ARRAY[1..GVL_CONSTANTS.C_MAX_MANIFOLDS] OF INT;  (* Аналоговые входы: Температура обратной линии (в 10-х долях градуса) *)
  AO_Supply_Fans : ARRAY[1..GVL_CONSTANTS.C_MAX_SUPPLY_FANS] OF UINT;  (* Аналоговые выходы: Скорость приточных вентиляторов (0-10В) *)
  AO_Exhaust_Fans : ARRAY[1..GVL_CONSTANTS.C_MAX_EXHAUST_FANS] OF UINT;  (* Аналоговые выходы: Скорость вытяжных вентиляторов (0-10В) *)
  AO_Lighting_Levels : ARRAY[1..GVL_CONSTANTS.C_MAX_ZONES] OF UINT;  (* Аналоговые выходы: диммирование освещения (0-1000 -> 0..100%) *)
  AO_Blinds_Positions : ARRAY[1..GVL_CONSTANTS.C_MAX_BLINDS] OF UINT;  (* Аналоговые выходы: позиционирование штор/жалюзи (0-1000 -> 0..100%) *)
  AI_Supply_Temps : ARRAY[1..GVL_CONSTANTS.C_MAX_SUPPLY_TEMPS] OF ST_Owen_Analog_Value;  (* Аналоговые входы: Температура приточного воздуха после калорифера *)
  AI_Boiler_Modulation : ARRAY[1..GVL_CONSTANTS.C_MAX_BOILERS] OF INT;  (* Аналоговые входы: Текущий уровень модуляции мощности котла (%) *)
  AI_Boiler_Flame_Status : ARRAY[1..GVL_CONSTANTS.C_MAX_BOILERS] OF BOOL;  (* Дискретные входы: Датчик ионизации (подтверждение наличия пламени) *)
  DI_Boiler_Error : ARRAY[1..GVL_CONSTANTS.C_MAX_BOILERS] OF BOOL;  (* Дискретные входы: Сигнал общей ошибки/аварии котла *)
  AI_Methane_LEL : ARRAY[1..GVL_CONSTANTS.C_MAX_METHANE_SENSORS] OF ST_Owen_Analog_Value;  (* Аналоговые входы: Уровень метана CH4 (0-100% LEL) *)
  AI_CO_PPM : ARRAY[1..GVL_CONSTANTS.C_MAX_CO_SENSORS] OF REAL;  (* Аналоговые входы: Уровень угарного газа CO (PPM) *)
  DI_Smoke_Sensors : ARRAY[1..GVL_CONSTANTS.C_MAX_SMOKE_SENSORS] OF BOOL;  (* Дискретные входы: Оптические датчики дыма (пожарный шлейф) *)
  AI_Temp_Outdoor : ST_Owen_Analog_Value;  (* Аналоговый вход: Наружная температура воздуха (уличный датчик) *)
  AI_Floor_Temps : ARRAY[1..GVL_CONSTANTS.C_MAX_ZONES] OF REAL;  (* Аналоговые входы: Температура стяжки пола по зонам (датчики в гильзах) *)
  AI_Room_Temps : ARRAY[1..GVL_CONSTANTS.C_MAX_ZONES] OF REAL;  (* Аналоговые входы: Температура воздуха в помещениях (настенные датчики) *)
  AI_Room_Hum : ARRAY[1..GVL_CONSTANTS.C_MAX_ZONES] OF REAL;  (* Аналоговые входы: Влажность воздуха в помещениях (%) *)
  AI_Room_CO2 : ARRAY[1..GVL_CONSTANTS.C_MAX_ZONES] OF REAL;  (* Аналоговые входы: Уровень CO2 в помещениях (ppm) *)
  DO_Zone_Valves : ARRAY[1..GVL_CONSTANTS.C_MAX_ZONES] OF BOOL;  (* Дискретные выходы: Термоэлектрические приводы контуров (220В) *)
  AI_DHW_Temp : REAL;  (* Аналоговый вход: Температура воды в бойлере косвенного нагрева *)
  AI_DHW_Pressure : REAL;  (* Аналоговый вход: Давление в контуре ГВС (контроль подпитки и утечек) *)
  DO_DHW_Heating_Pump : BOOL;  (* Дискретный выход: Насос загрузки бойлера (первичный контур от котла) *)
  DO_DHW_Circ_Pump : BOOL;  (* Дискретный выход: Насос рециркуляции ГВС (кольцо потребителей) *)
  DO_Backup_Circulation_Pump : BOOL;  (* Дискретный выход: Резервный циркуляционный насос антизамерзания *)
  DO_Electric_Heater_Enable : BOOL;  (* Дискретный выход: Сухой контакт электрического нагревателя антизамерзания *)
  DI_Lighting_Switches : ARRAY[1..GVL_CONSTANTS.C_MAX_ZONES] OF BOOL;  (* Дискретные входы: Физические кнопки/выключатели (импульсные) *)
  DI_Socket_Switches : ARRAY[1..GVL_CONSTANTS.C_MAX_SOCKETS] OF BOOL;  (* Legacy-вход: локальные выключатели розеток отключены концептуально *)
  DI_Motion_Sensors : ARRAY[1..GVL_CONSTANTS.C_MAX_ZONES] OF BOOL;  (* Дискретные входы: Датчики присутствия (PIR-сенсоры) *)
  DO_Sockets : ARRAY[1..GVL_CONSTANTS.C_MAX_SOCKETS] OF BOOL;  (* Дискретные выходы: Управление розетками (реле) *)
  DO_Gas_Valve_Close : BOOL;  (* Дискретный выход: Импульс на закрытие электромагнитного газового клапана *)
  DO_Water_Valve_35_Close : BOOL;  (* Дискретный выход: Закрыть вводной шаровый кран воды №1 (с электроприводом) *)
  DO_Water_Valve_36_Close : BOOL;  (* Дискретный выход: Закрыть вводной шаровый кран воды №2 (с электроприводом) *)
  AI_Water_Valve_35_Current : REAL;  (* Аналоговый вход: Ток потребления электропривода крана №1 (контроль заклинивания) *)
  AI_Water_Valve_36_Current : REAL;  (* Аналоговый вход: Ток потребления электропривода крана №2 (контроль заклинивания) *)
  DI_Power_OK : BOOL;  (* Дискретный вход: Контроль наличия напряжения на вводе (реле контроля фаз) *)
  DO_Gas_Siren : BOOL;  (* Дискретный выход: Звуковое оповещение при опасной концентрации газа *)
  DO_Fire_Siren : BOOL;  (* Дискретный выход: Звуковое оповещение при обнаружении задымления *)
  DO_Security_Siren : BOOL;  (* Дискретный выход: Сирена охранной сигнализации *)
  DO_Pump_Main_Enable : BOOL;  (* Дискретный выход: Разрешение работы главного циркуляционного насоса системы *)
  DO_Gate_Open : BOOL;  (* Дискретный выход: Команда на открытие въездных ворот (импульс) *)
  DO_Wicket_Open : BOOL;  (* Дискретный выход: Команда на разблокировку электрозамка калитки *)
  DO_Lock_1_Open : BOOL;  (* Дискретный выход: Разблокировать основной электромеханический замок дома *)
  DO_Lock_1_Close : BOOL;  (* Дискретный выход: Заблокировать основной электромеханический замок дома *)
  DO_Lock_2_Open : BOOL;  (* Дискретный выход: Разблокировать дополнительный замок (черный ход) *)
  DO_Lock_2_Close : BOOL;  (* Дискретный выход: Заблокировать дополнительный замок (черный ход) *)
  DI_Partner_Pulse : BOOL;  (* Дискретный вход: Пульс от второго ПЛК *)
  DI_Partner_Active : BOOL;  (* Дискретный вход: Статус активности второго ПЛК *)
  DO_Heartbeat_Pulse : BOOL;  (* Дискретный выход: Собственный пульс *)
  DO_Active_Status : BOOL;  (* Дискретный выход: Собственный статус активности *)
  DI_Module_1_Heartbeat : BOOL;  (* Сигнал жизни от модуля 1 *)
  DI_Module_2_Heartbeat : BOOL;  (* Сигнал жизни от модуля 2 *)
  DI_Backup_Circulation_Pump_Feedback : BOOL;  (* Обратная связь резервного циркуляционного насоса *)
  DI_Electric_Heater_Feedback : BOOL;  (* Обратная связь электрического нагревателя *)
  DI_Water_Zone_Open_FB : ARRAY[1..32] OF BOOL;  (* Концевики: зональный водяной клапан открыт *)
  DI_Water_Zone_Close_FB : ARRAY[1..32] OF BOOL;  (* Концевики: зональный водяной клапан закрыт *)
  DO_Water_Zone_Enable : ARRAY[1..32] OF BOOL;  (* Разрешение подачи воды по зонам *)
END_VAR

VAR_GLOBAL RETAIN  (* GVL_PERSISTENT *)
  P_System_Mode : E_System_Operating_Mode;
  P_Safety_Gas_Latched : BOOL;
  P_Safety_Smoke_Latched : BOOL;
  P_Safety_Leak_Latched : BOOL;
  P_DHW_Heating_Active : BOOL;
  P_Valid : BOOL;
END_VAR

VAR_GLOBAL  (* GVL_COMMAND_SHADOW *)
  G_Gas_Valve_Close : BOOL := FALSE;
  G_Boiler_Stop : BOOL := FALSE;
  G_Supply_100_Req : BOOL := FALSE;
  G_Supply_80_Req : BOOL := FALSE;
  G_Vent_PV3_Boost : BOOL := FALSE;
  G_Exhaust_100_Req : BOOL := FALSE;
  G_Vent_Stop : BOOL := FALSE;
  G_Close_Valve_35 : BOOL := FALSE;
  G_Close_Valve_36 : BOOL := FALSE;
  G_Lock_1_Open : BOOL := FALSE;
  G_Lock_1_Close : BOOL := FALSE;
  G_Lock_2_Open : BOOL := FALSE;
  G_Lock_2_Close : BOOL := FALSE;
  G_Gate_Open : BOOL := FALSE;
  G_Wicket_Open : BOOL := FALSE;
END_VAR

{attribute 'qualified_only'}
VAR_GLOBAL  (* GVL_TEST_PANEL_DEBUG *)
  G_Test_Description : STRING(200);
  G_Test_What_To_Change : STRING(200);
  G_Test_Expected_Text : STRING(200);
  G_Expected_Summary : STRING(200);
  G_Actual_Summary : STRING(200);
  G_Error_Text : STRING(200);
  G_System_State_Line : STRING(200);
  G_Input_Guest_Preheat_Request : BOOL;
  G_Input_Guest_Preheat_Enabled : BOOL;
  G_Input_Guest_Preheat_Boost : INT;
  G_Input_Max_Thermal_Budget : REAL;
  G_Input_Block_Heating : BOOL;
  G_Input_Safety_Stop : BOOL;
END_VAR

{attribute 'qualified_only'}
VAR_GLOBAL  (* GVL_MODE *)
  G_Current_Behavior_Mode : E_Behavior_Mode := BEHAVIOR_HOME;
  G_Mode_Last_Change_TS : UDINT := 0;
  G_Mode_Code : UDINT := 0;
  G_Away_Request : BOOL := FALSE;
  G_Maintenance_Request : BOOL := FALSE;
END_VAR

VAR_GLOBAL  (* GVL_Safety_Selector *)
  G_Use_Shadow_CO : BOOL := FALSE;
  G_Use_Shadow_Methane : BOOL := FALSE;
  G_Use_Shadow_Smoke : BOOL := FALSE;
  G_CO_Effective : REAL;
  G_Methane_Effective : REAL;
  G_Smoke_Effective : BOOL;
  G_CO_Shadow_Max_Diff : REAL := 5.0;
  G_Methane_Shadow_Max_Diff : REAL := 5.0;
  G_Block_Shadow_On_Mismatch : BOOL := TRUE;
  G_Shadow_Unstable_Cycles_Limit : INT := 5;
  G_CO_Shadow_Recovery_Diff : REAL := 2.0;
  G_Methane_Shadow_Recovery_Diff : REAL := 2.0;
  G_CO_Stable_Counter : INT := 0;
  G_Methane_Stable_Counter : INT := 0;
  G_Smoke_Stable_Counter : INT := 0;
  G_CO_Unstable_Counter : INT := 0;
  G_Methane_Unstable_Counter : INT := 0;
  G_Smoke_Unstable_Counter : INT := 0;
  G_CO_Effective_Array : ARRAY[1..GVL_CONSTANTS.C_MAX_CO_SENSORS] OF REAL;
  G_Methane_Effective_Array : ARRAY[1..GVL_CONSTANTS.C_MAX_METHANE_SENSORS] OF REAL;
  G_Smoke_Effective_Array : ARRAY[1..GVL_CONSTANTS.C_MAX_SMOKE_SENSORS] OF BOOL;
END_VAR

{attribute 'qualified_only'}
VAR_GLOBAL  (* GVL_TEST *)
  G_Test_Enable : BOOL := FALSE;
  G_Test_Total_Checks : INT := 0;
  G_Test_Failed_Checks : INT := 0;
  G_Test_Passed : BOOL := TRUE;
  G_Test_Last_Failure_Index : INT := 0;
  G_Test_Last_Failure_Code : UDINT := 0;
  G_Test_Status_Msg : STRING(200) := 'Tests not run';
  G_Ownership_Violation : BOOL := FALSE;
  G_Diagnostics_Duplicate_Event_Found : BOOL := FALSE;
  G_Diagnostics_Count_Out_Of_Range : BOOL := FALSE;
  G_Heating_Allocation_Budget_Exceeded : BOOL := FALSE;
  G_Heating_Allocation_Enabled_Not_Allowed : BOOL := FALSE;
  G_Safety_Latched_Without_Intent : BOOL := FALSE;
  G_HP_Adjusted_Priority_Lower_Bound_Violation : BOOL := FALSE;
  G_HP_Adjusted_Allocation_Budget_Exceeded : BOOL := FALSE;
  G_HP_Adjusted_Allocation_Enabled_Not_Allowed : BOOL := FALSE;
  G_HP_Guest_Preheat_Config_Out_Of_Range : BOOL := FALSE;
  G_HP_Manifold_Adjusted_Priority : ARRAY[1..GVL_CONSTANTS.C_MAX_MANIFOLDS] OF INT;
END_VAR

{attribute 'qualified_only'}
VAR_GLOBAL  (* GVL_HEATING_POLICY *)
  G_Zone_Empty_Duration_MS : ARRAY[1..GVL_CONSTANTS.C_MAX_ZONES] OF UDINT;
  G_Zone_Permanent_Use : ARRAY[1..GVL_CONSTANTS.C_MAX_ZONES] OF BOOL;
  G_Zone_Guest_Preheat_Request : ARRAY[1..GVL_CONSTANTS.C_MAX_ZONES] OF BOOL;
  G_Zone_Policy_Class : ARRAY[1..GVL_CONSTANTS.C_MAX_ZONES] OF INT;
  G_Zone_Target_Adjustment : ARRAY[1..GVL_CONSTANTS.C_MAX_ZONES] OF REAL;
  G_Zone_Priority_Bias : ARRAY[1..GVL_CONSTANTS.C_MAX_ZONES] OF REAL;
END_VAR

{attribute 'qualified_only'}
VAR_GLOBAL  (* GVL_GATEWAY *)
  G_Gateway_Command : ST_Gateway_Command;
  G_Gateway_Command_Received : BOOL;
  G_Gateway_Send_2FA : BOOL;
  G_Gateway_2FA_Code : STRING(6);
  G_Gateway_Telegram_Msg : STRING(200);
  G_Gateway_Send_Telegram : BOOL;
  G_Gateway_HMI_Status_Message : STRING(200);
  G_Gateway_Ping_OK : BOOL;
  G_Gateway_Data_Ready : BOOL;
  G_Gateway_Modbus_Registers : ARRAY[0..GVL_CONSTANTS.C_MAX_MODBUS_REGISTERS-1] OF WORD;
  G_Shadow_Alert_Active : BOOL;
  G_Shadow_Dominant_Channel : STRING(32);
  G_Shadow_Policy_Summary_Text : STRING(160);
  G_Shadow_Recent_Activity_Text : STRING(160);
  G_Shadow_Rate_Summary_Text : STRING(160);
  G_Shadow_Total_Fallback_Count : UDINT;
  G_Shadow_Total_Recovery_Count : UDINT;
END_VAR

VAR_GLOBAL  (* GVL_EVENT *)
  G_Event_Log : ARRAY[0..63] OF ST_EVENT;
  G_Event_Head : UINT;
  G_Event_ID_Counter : UDINT;
END_VAR

{attribute 'qualified_only'}
VAR_GLOBAL  (* GVL_PRESENCE *)
  G_Any_Motion : BOOL := FALSE;
  G_Occupied : BOOL := TRUE;
  G_Auto_Away_Request : BOOL := FALSE;
  G_Last_Motion_TS : UDINT := 0;
  G_Zone_Occupied : ARRAY[1..GVL_CONSTANTS.C_MAX_ZONES] OF BOOL;
  G_Zone_Last_Motion_TS : ARRAY[1..GVL_CONSTANTS.C_MAX_ZONES] OF UDINT;
END_VAR

{attribute 'qualified_only'}
VAR_GLOBAL  (* GVL_STATE *)
  G_Floor_Temps : ARRAY[1..GVL_CONSTANTS.C_MAX_HEATING_CIRCUITS] OF REAL;  (* Массив текущих температур поверхности пола по физическим контурам *)
  G_Room_Temps : ARRAY[1..GVL_CONSTANTS.C_MAX_ZONES] OF REAL;
  G_Room_Hum : ARRAY[1..GVL_CONSTANTS.C_MAX_ZONES] OF REAL;
  G_Room_CO2 : ARRAY[1..GVL_CONSTANTS.C_MAX_ZONES] OF REAL;
  G_Motion_Sensors : ARRAY[1..32] OF BOOL;
  G_Door_Sensors : ARRAY[1..GVL_CONSTANTS.C_MAX_DOOR_SENSORS] OF BOOL;
  G_Window_Sensors : ARRAY[1..GVL_CONSTANTS.C_MAX_ZONES] OF BOOL;
  G_Water_Sensors : ARRAY[1..GVL_CONSTANTS.C_MAX_FLOOD_SENSORS] OF BOOL;
  G_Smoke_Sensors : ARRAY[1..GVL_CONSTANTS.C_MAX_SMOKE_SENSORS] OF BOOL;
  G_Methane_Sensors : ARRAY[1..GVL_CONSTANTS.C_MAX_METHANE_SENSORS] OF REAL;
  G_CO_Sensors : ARRAY[1..GVL_CONSTANTS.C_MAX_CO_SENSORS] OF REAL;
  G_Manifold_Pressures : ARRAY[1..GVL_CONSTANTS.C_MAX_MANIFOLDS] OF REAL;
  G_Manifold_Currents : ARRAY[1..GVL_CONSTANTS.C_MAX_MANIFOLDS] OF REAL;
  G_Manifold_T_Supply : ARRAY[1..GVL_CONSTANTS.C_MAX_MANIFOLDS] OF REAL;
  G_Manifold_T_Return : ARRAY[1..GVL_CONSTANTS.C_MAX_MANIFOLDS] OF REAL;
  G_Boiler_Flame : ARRAY[1..GVL_CONSTANTS.C_MAX_BOILERS] OF BOOL;
  G_Boiler_Error : ARRAY[1..GVL_CONSTANTS.C_MAX_BOILERS] OF BOOL;
  G_Boiler_OT_Online : ARRAY[1..GVL_CONSTANTS.C_MAX_BOILERS] OF BOOL;  (* Статус доступности OpenTherm-канала котла от реального OT-адаптера/драйвера *)
  G_Boiler_OT_Enable : ARRAY[1..GVL_CONSTANTS.C_MAX_BOILERS] OF BOOL;  (* Команды разрешения через OpenTherm *)
  G_Boiler_OT_Setpoint : ARRAY[1..GVL_CONSTANTS.C_MAX_BOILERS] OF REAL;  (* Уставки через OpenTherm *)
  G_Physical_Switches : ARRAY[1..32] OF BOOL;
  G_Socket_Switches : ARRAY[1..GVL_CONSTANTS.C_MAX_SOCKETS] OF BOOL;  (* Legacy-поле: локальные выключатели розеток не используются *)
  G_Outdoor_Temp : REAL;
  G_Supply_Temps : ARRAY[1..GVL_CONSTANTS.C_MAX_SUPPLY_TEMPS] OF REAL;  (* Температура приточного воздуха после калорифера *)
  G_DHW_Temp : REAL;
  G_DHW_Pressure : REAL;
  G_Zone_Valves : ARRAY[1..GVL_CONSTANTS.C_MAX_HEATING_CIRCUITS] OF BOOL;
  G_Manifold_Pumps : ARRAY[1..GVL_CONSTANTS.C_MAX_MANIFOLDS] OF BOOL;
  G_Manifold_Valves : ARRAY[1..GVL_CONSTANTS.C_MAX_MANIFOLDS] OF REAL;  (* 0.0 - 1.0 *)
  G_Manifold_End_Switches : ARRAY[1..GVL_CONSTANTS.C_MAX_MANIFOLDS] OF BOOL;  (* Концевики клапанов *)
  G_Supply_Fans : ARRAY[1..GVL_CONSTANTS.C_MAX_SUPPLY_FANS] OF REAL;  (* 0.0 - 1.0 *)
  G_Exhaust_Fans : ARRAY[1..GVL_CONSTANTS.C_MAX_EXHAUST_FANS] OF REAL;  (* 0.0 - 1.0 *)
  G_Vent_Heater_Power : ARRAY[1..GVL_CONSTANTS.C_MAX_BOILERS] OF REAL;
  G_Lighting_Levels : ARRAY[1..32] OF BYTE;
  G_Blinds_Positions : ARRAY[1..GVL_CONSTANTS.C_MAX_BLINDS] OF BYTE;
  G_Socket_States : ARRAY[1..GVL_CONSTANTS.C_MAX_SOCKETS] OF BOOL;
  G_DHW_Heating_Pump : BOOL;
  G_DHW_Circ_Pump : BOOL;
  G_Backup_Circulation_Pump : BOOL;  (* Резервный циркуляционный насос для антизамерзания при газовой аварии *)
  G_Electric_Heater_Enable : BOOL;  (* Сухой контакт электрического нагревателя для антизамерзания *)
  G_Safety_Gas_Alarm : BOOL;
  G_Safety_Leak_Alarm : BOOL;
  G_Safety_Smoke_Alarm : BOOL;
  G_Safety_Emergency_Stop : BOOL;  (* агрегированный аварийный стоп *)
  G_Safety_Gas_Latched : BOOL;  (* защёлкнутая газовая авария *)
  G_Safety_Leak_Latched : BOOL;  (* защёлкнутая авария протечки *)
  G_Safety_Smoke_Latched : BOOL;  (* защёлкнутая дымовая/пожарная авария *)
  G_Safety_Freeze_Risk : BOOL;  (* риск замерзания при защёлкнутой газовой аварии *)
  G_System_Mode : E_System_Operating_Mode := E_System_Operating_Mode.MODE_NORMAL;  (* Текущий режим работы системы *)
  G_System_Mode_Text : STRING(64);
  G_Heating_IO_Fault : BOOL;
  G_Heating_Sensor_Fault : BOOL;
  G_Heating_Subsystem_Degraded : BOOL;
  G_DHW_IO_Fault : BOOL;
  G_DHW_Sensor_Fault : BOOL;
  G_DHW_Subsystem_Degraded : BOOL;
  G_Ventilation_IO_Fault : BOOL;
  G_Ventilation_Subsystem_Degraded : BOOL;
  G_Lighting_IO_Fault : BOOL;
  G_Lighting_Subsystem_Degraded : BOOL;
  G_Access_Comm_Fault : BOOL;
  G_Evacuation_Lighting_Active : BOOL;
  G_Evac_Hazard_Zone : ARRAY[1..32] OF BOOL;  (* опасные зоны (дым/протечка) *)
  G_Evac_Guidance : ARRAY[1..32] OF INT;  (* -1 = избегать, 0 = нейтрально, +1 = к выходу *)
  G_Rule_Actions : ARRAY[1..GVL_CONSTANTS.C_MAX_RULES] OF ST_Rule_Action;
  G_Sim_Lights : ARRAY[1..32] OF BOOL;
  G_Freeze_Hardware_Degraded : BOOL;  (* Деградация anti-freeze hardware *)
  G_Freeze_Hardware_Failed : BOOL;  (* Критический отказ anti-freeze hardware *)
  G_Water_Zone_Enable : ARRAY[1..32] OF BOOL;  (* Селективное открытие воды по зонам *)
  G_Water_Zone_Open_FB : ARRAY[1..32] OF BOOL;  (* Обратная связь: зональный клапан открыт *)
  G_Water_Zone_Close_FB : ARRAY[1..32] OF BOOL;  (* Обратная связь: зональный клапан закрыт *)
  G_Water_Zone_Exercise_Active : ARRAY[1..32] OF BOOL;  (* Профилактическая прокрутка шаровых кранов *)
  G_Preheat_Request : BOOL;  (* Heating request: preheat *)
  G_Freeze_Request : BOOL;  (* Heating request: freeze *)
  G_Target_Temperature : REAL;  (* Heating arbitration target *)
END_VAR

VAR_GLOBAL  (* GVL_INTENT_USER *)
  I_Source_Valid : BOOL := FALSE;
  I_Last_Update_Cycle : UDINT := 0;
  I_Last_Update_MS : UDINT := 0;
  I_Arm_Request : BOOL := FALSE;
  I_Disarm_Request : BOOL := FALSE;
  I_PIN_Code : STRING(8);
  I_RFID_Tag : STRING(32);
  I_2FA_Code_In : STRING(8);
  I_Gate_Open_Request : BOOL := FALSE;
  I_Wicket_Open_Request : BOOL := FALSE;
  I_Lock_1_Open_Request : BOOL := FALSE;
  I_Lock_1_Close_Request : BOOL := FALSE;
  I_Lock_2_Open_Request : BOOL := FALSE;
  I_Lock_2_Close_Request : BOOL := FALSE;
  I_Dangerous_Action_Request : BOOL := FALSE;
  I_Dangerous_Action_Confirm : BOOL := FALSE;
  I_User_Access_Level : INT := 0;
  I_Water_Valve_Test_Open : BOOL := FALSE;
  I_Water_Valve_Test_Close : BOOL := FALSE;
  I_Water_Valve_Test_Confirm : BOOL := FALSE;
  I_Gas_Valve_Test_Open : BOOL := FALSE;
  I_Gas_Valve_Test_Close : BOOL := FALSE;
  I_Gas_Valve_Test_Confirm : BOOL := FALSE;
  I_Water_Selective_Recover : BOOL := FALSE;
  I_Gas_Selective_Recover : BOOL := FALSE;
  I_Scenario_Request : E_SCENARIO_TYPE := E_SCENARIO_TYPE.SCENARIO_NONE;
  I_Lighting_Override_32 : ARRAY[1..32] OF BYTE;
  I_Blinds_Override_32 : ARRAY[1..GVL_CONSTANTS.C_MAX_BLINDS] OF BYTE;
  I_Socket_Override_32 : ARRAY[1..GVL_CONSTANTS.C_MAX_SOCKETS] OF BOOL;
  I_Reset_Errors : BOOL := FALSE;
  I_Set_Temp_Req : BOOL := FALSE;
  I_Target_Zone : INT := 0;
  I_Target_Temperature : REAL := 0.0;
  I_Set_Vent_Req : BOOL := FALSE;
  I_Target_Vent_Speed : REAL := 0.0;
  I_Set_Config_Req : BOOL := FALSE;
  I_Time_Sync_Req : BOOL := FALSE;
  I_New_Time_MS : UDINT := 0;
END_VAR

{attribute 'qualified_only'}
VAR_GLOBAL  (* GVL_STATUS *)
  G_System_Time_MS : UDINT;  (* Системное время в миллисекундах *)
  G_Last_System_Time_MS : UDINT := 0;  (* Предыдущее системное время (для детекции переполнения) *)
  G_Time_Of_Day_MS : UDINT := 0;  (* Время от начала суток в мс (0-86399999) *)
  G_Current_Day : UINT := 1;  (* Текущий день недели (1-7) *)
  G_Day_Of_Year : UINT := 1;  (* Текущий день года (1-365) *)
  G_Current_TOD : TOD;  (* Текущее время суток *)
  G_Current_Scenario : E_SCENARIO_TYPE := E_SCENARIO_TYPE.SCENARIO_NONE;  (* Текущий активный сценарий *)
  G_Previous_Scenario : E_SCENARIO_TYPE := E_SCENARIO_TYPE.SCENARIO_NONE;  (* Предыдущий сценарий *)
  G_Is_Night : BOOL;  (* Флаг ночного времени *)
  G_PLC_ID : BYTE := 1;  (* 1 = PLC_A, 2 = PLC_B *)
  G_Is_Active_PLC : BOOL;
  G_Local_PLC_ID : BYTE := 1;  (* Идентификатор данного ПЛК в паре *)
  G_Active_PLC_ID : BYTE := 1;  (* Идентификатор ведущего ПЛК *)
  G_Remote_PLC_Pulse : BOOL;  (* Сигнал "жизни" от второго ПЛК *)
  G_Security_Status_Msg : STRING(200);
  G_Gas_Status_Msg : STRING(200);
  G_Flood_Status_Msg : STRING(200);
  G_Vent_Status_Msg : STRING(200);
  G_DHW_Status : ST_DHW_Status;
  G_Manifold_Status : ARRAY[1..GVL_CONSTANTS.C_MAX_MANIFOLDS] OF ST_Manifold_Status;
  G_Boiler_Status : ARRAY[1..GVL_CONSTANTS.C_MAX_BOILERS] OF ST_Boiler_Status;
  G_IO_Modules_Online : ARRAY[1..GVL_CONSTANTS.C_MAX_MODULES] OF BOOL;  (* Статусы модулей ввода-вывода *)
  G_Sim_Active : BOOL;
  G_Wet_Zone_Light_Active : BOOL;
  G_System_Mode_Msg : STRING(200);  (* Пояснение текущего режима работы системы для HMI *)
  G_System_Mode_Cause : STRING(200);  (* Корневая причина режима (пожар/газ/протечка/штатно) *)
  G_Evac_Target_Zone_Name : STRING(80);  (* Предпочтительная зона выхода/направления эвакуации *)
  G_Evac_Hazard_Zone_Name : STRING(80);  (* Наиболее важная опасная зона для HMI/диагностики *)
  G_Diagnostics : ST_System_Diagnostics;  (* Интегральная диагностика и HMI-состояния *)
  G_Diagnostics_Events : ARRAY[1..50] OF ST_Diagnostic_Event;
  G_Diagnostics_Count : INT := 0;
END_VAR

{attribute 'qualified_only'}
VAR_GLOBAL  (* GVL_ALARM *)
  G_Security_Armed : BOOL := FALSE;  (* Флаг: Система безопасности активирована *)
  G_Security_Siren : BOOL := FALSE;
  G_Global_Siren : BOOL := FALSE;  (* Глобальный флаг сирены от Alarm Manager *)
  G_Global_Critical : BOOL := FALSE;
  G_Global_Warning : BOOL := FALSE;
  G_Active_Alarm_Count : INT := 0;
  G_Unacked_Alarm_Count : INT := 0;
  G_Alarm_List : ARRAY[1..GVL_CONSTANTS.C_MAX_ALARMS] OF ST_Alarm_Record;
  G_Gas_Alarm_Active : BOOL := FALSE;  (* Флаг: Обнаружена критическая концентрация газа *)
  G_Gas_Fire_Siren : BOOL := FALSE;
  G_Fire_Alarm_Active : BOOL := FALSE;  (* Флаг: Сработали пожарные датчики *)
  G_Flood_Alarm_Active : BOOL := FALSE;  (* Флаг: Обнаружена протечка воды *)
  G_Security_Alarm : BOOL := FALSE;  (* Флаг: Тревога системы безопасности *)
END_VAR

{attribute 'qualified_only'}
VAR_GLOBAL  (* GVL_HEATING_POLICY_CONFIG *)
  G_Guest_Preheat_Enabled : BOOL := TRUE;
  G_Guest_Preheat_Priority_Boost : INT := 2;
  G_Guest_Preheat_Max_Duration_MS : UDINT := 7200000;  (* 2 hours (future use) *)
END_VAR

{attribute 'qualified_only'}
VAR_GLOBAL  (* GVL_CONFIG *)
  G_Heating_Config : ST_Heating_Config;  (* Настройки системы отопления *)
  G_Ventilation_Config : ST_Ventilation_Config;  (* Настройки системы вентиляции *)
  G_DHW_Config : ST_DHW_Config;  (* Настройки горячего водоснабжения *)
  G_Security_Config : ST_Security_Global_Config;  (* Настройки системы безопасности *)
  G_Flood_Config : ST_Flood_Config;  (* Настройки системы защиты от протечек *)
  G_HMI_FloorHeating_Configs : ARRAY[1..GVL_CONSTANTS.C_MAX_HEATING_CIRCUITS] OF ST_FloorHeating_Circuit_Config;  (* Конфигурации контуров теплого пола *)
  G_Heating_Circuit_To_Zone : ARRAY[1..GVL_CONSTANTS.C_MAX_HEATING_CIRCUITS] OF INT := [1, 2, 3, 4, 5, 6, 7, 8, 9, 10, 11, 12, 13, 14, 15, 16];  (* ВРЕМЕННО: circuit -> zone mapping, требует уточнения по фактической таблице помещений *)
  G_Wet_Zone_Map : ARRAY[1..32] OF BOOL;  (* Карта мокрых зон (TRUE = мокрая зона) *)
  G_HMI_Tariff_Settings : ST_Tariff_Config;  (* Настройки тарифов *)
  G_HMI_Vent_Global_Config : ST_Ventilation_Global_Config;  (* Глобальные настройки вентиляции *)
  G_HMI_Vent_Unit_Configs : ARRAY[1..GVL_CONSTANTS.C_MAX_VENT_UNITS] OF ST_Ventilation_Unit_Config;  (* Конфигурации отдельных вентустановок *)
  G_HMI_Scenario_Configs : ARRAY[1..GVL_CONSTANTS.C_MAX_SCENARIOS] OF ST_Scenario_Config;  (* Конфигурации сценариев *)
  G_HMI_Outdoor_Configs : ARRAY[1..GVL_CONSTANTS.C_MAX_OUTDOOR_ZONES] OF ST_Outdoor_Zone_Config;  (* Конфигурации зон уличного освещения *)
  G_HMI_Flood_Config : ST_Flood_Global_Config;  (* Глобальные настройки защиты от протечек *)
  G_HMI_Gas_Config : ST_Gas_Valve_Configuration;  (* Конфигурация системы газового контроля *)
  G_HMI_Sensor_Calibrations : ARRAY[1..GVL_CONSTANTS.C_MAX_CALIBRATIONS] OF ST_Sensor_Calibration_Record;  (* Данные калибровки датчиков *)
  G_HMI_User_Rules : ARRAY[1..GVL_CONSTANTS.C_MAX_RULES] OF ST_User_Rule;  (* Пользовательские правила (Rule Engine) *)
  G_Enable_Sensor_Calibration : BOOL := TRUE;
  G_Calib_Outdoor_Temp : ST_Sensor_Calibration_Record;
  G_Calib_Supply_Temps : ARRAY[1..GVL_CONSTANTS.C_MAX_SUPPLY_TEMPS] OF ST_Sensor_Calibration_Record;
  G_Calib_Room_Temps : ARRAY[1..GVL_CONSTANTS.C_MAX_ZONES] OF ST_Sensor_Calibration_Record;
  G_Calib_Floor_Temps : ARRAY[1..GVL_CONSTANTS.C_MAX_ZONES] OF ST_Sensor_Calibration_Record;
  G_Calib_CO2 : ARRAY[1..GVL_CONSTANTS.C_MAX_ZONES] OF ST_Sensor_Calibration_Record;
  G_Calib_Humidity : ARRAY[1..GVL_CONSTANTS.C_MAX_ZONES] OF ST_Sensor_Calibration_Record;
  G_Calib_Manifold_T_Supply : ARRAY[1..GVL_CONSTANTS.C_MAX_MANIFOLDS] OF ST_Sensor_Calibration_Record;
  G_Calib_Manifold_T_Return : ARRAY[1..GVL_CONSTANTS.C_MAX_MANIFOLDS] OF ST_Sensor_Calibration_Record;
  G_Calib_Methane : ARRAY[1..GVL_CONSTANTS.C_MAX_METHANE_SENSORS] OF ST_Sensor_Calibration_Record;
  G_Calib_CO : ARRAY[1..GVL_CONSTANTS.C_MAX_CO_SENSORS] OF ST_Sensor_Calibration_Record;
  G_Valve_Test_Config : ARRAY[1..GVL_CONSTANTS.C_MAX_MANIFOLDS] OF ST_Valve_Test_Config;
  G_HMI_Cleaning_Mode_Active : ARRAY[1..GVL_CONSTANTS.C_MAX_CLEANING_MODES] OF BOOL;  (* Режим уборки активен *)
  G_HMI_Cleaning_Mode_TimeLeft : ARRAY[1..GVL_CONSTANTS.C_MAX_CLEANING_MODES] OF UINT;  (* Оставшееся время режима уборки *)
  G_HMI_Admin_2FA_Enabled : BOOL := FALSE;  (* Включена ли 2FA для ADMIN *)
  G_HMI_Current_Operator_Factor2_Done : BOOL;  (* Второй фактор пройден *)
  G_HMI_Current_Operator_ID : STRING(10);  (* ID текущего оператора *)
  G_HMI_Manual_Gas_Valve_Open : BOOL;  (* Ручное открытие газового клапана *)
  G_HMI_Manual_Gas_Valve_Time : UDINT := 5;  (* Время ручного открытия *)
  G_HMI_Manual_Gas_Valve_TimeLeft : UDINT;  (* Оставшееся время ручного открытия *)
  G_HMI_Apply_Settings : BOOL;  (* Команда: Применить настройки *)
  G_HMI_Mute_Alarm : BOOL;  (* Команда: Временное отключение сирены *)
  G_HMI_Ack_Alarms : BOOL;  (* Команда: Квитировать все тревоги *)
  G_HMI_Gate_Open_Req : BOOL;  (* Запрос на открытие въездных ворот *)
  G_HMI_Wicket_Open_Req : BOOL;  (* Запрос на открытие калитки *)
  G_HMI_Lock_1_Open_Req : BOOL;  (* Разблокировка основного замка *)
  G_HMI_Lock_1_Close_Req : BOOL;  (* Блокировка основного замка *)
  G_HMI_Lock_2_Open_Req : BOOL;  (* Разблокировка доп. замка *)
  G_HMI_Lock_2_Close_Req : BOOL;  (* Блокировка доп. замка *)
  G_HMI_Language : BYTE := 0;  (* 0=RU, 1=EN *)
  G_HMI_Brightness : BYTE := 80;
  G_HMI_Screen_Saver_Timeout : UDINT := 300;  (* сек *)
  G_Allowed_IPs : ARRAY[1..GVL_CONSTANTS.C_MAX_ALLOWED_IPS] OF STRING(15) := ['192.168.1.100', '192.168.1.101', '127.0.0.1', '', ''];  (* Разрешенные IP-адреса для шлюза *)
  G_Backup_Circulation_Pump_In_Service : BOOL := TRUE;  (* Резервный насос доступен для логики *)
  G_Electric_Heater_In_Service : BOOL := TRUE;  (* Электронагреватель доступен для логики *)
  G_Freeze_Hardware_Retry_Count : INT := 2;  (* Количество повторных попыток для anti-freeze hardware *)
  G_Freeze_Hardware_Retry_Delay_MS : UDINT := 5000;  (* Задержка между попытками повторного пуска *)
  G_Pump_Exercise_Enabled : BOOL := TRUE;  (* Разрешение периодической прокрутки насосов после простоя *)
  G_Pump_Exercise_Interval_MS : UDINT := 604800000;  (* 7 суток *)
  G_Pump_Exercise_Duration_MS : UDINT := 30000;  (* 30 сек *)
  G_Manifold_Pump_In_Service : ARRAY[1..GVL_CONSTANTS.C_MAX_MANIFOLDS] OF BOOL := [TRUE, TRUE, TRUE, TRUE, TRUE];
  G_Manifold_Priority : ARRAY[1..GVL_CONSTANTS.C_MAX_MANIFOLDS] OF INT := [3, 3, 2, 2, 1];  (* 3=high, 2=normal, 1=low *)
  G_Manifold_Thermal_Weight : ARRAY[1..GVL_CONSTANTS.C_MAX_MANIFOLDS] OF REAL := [1.0, 1.0, 0.8, 0.8, 0.5];
  G_Max_Active_Manifolds : INT := 3;  (* energy-management limit for simultaneous active manifolds *)
  G_Max_Thermal_Budget : REAL := 6.0;  (* simplified manifold thermal budget units *)
  G_DHW_Heating_Pump_In_Service : BOOL := TRUE;
  G_DHW_Circ_Pump_In_Service : BOOL := TRUE;
  G_Water_Valve_Exercise_Enabled : BOOL := TRUE;
  G_Water_Valve_Exercise_Interval_MS : UDINT := 604800000;
  G_Water_Valve_Exercise_Duration_MS : UDINT := 15000;
  G_Water_Valve_Exercise_Window_Start : TOD := TOD#04:00;
  G_Water_Valve_Exercise_Window_End : TOD := TOD#05:00;
  G_Water_Valve_Close_Retry_Count : INT := 2;
  G_Water_Valve_Close_Retry_Delay_MS : UDINT := 3000;
  G_FloorTemp_Map : ARRAY[1..GVL_CONSTANTS.C_MAX_HEATING_CIRCUITS] OF INT := [1, 2, 3, 4, 5, 6, 7, 8, 9, 10, 11, 12, 13, 14, 15, 16];
  G_RoomTemp_Map : ARRAY[1..16] OF INT := [1, 2, 3, 4, 5, 6, 7, 8, 9, 10, 11, 12, 13, 14, 15, 16];
  G_Door_Map : ARRAY[1..GVL_CONSTANTS.C_MAX_DOOR_SENSORS] OF INT := [1, 2, 3, 4, 5, 6, 7, 8];
  G_Window_Map : ARRAY[1..16] OF INT := [9, 10, 11, 12, 13, 14, 15, 16, 17, 18, 19, 20, 21, 22, 23, 24];
  C_MAX_LIGHT_ZONES : INT := 32;  (* fallback if not defined elsewhere *)
  G_Evac_Exit_Zones : ARRAY[1..32] OF BOOL;  (* зоны-выходы (TRUE = выход) *)
  G_Evac_Smoke_Zone_Map : ARRAY[1..GVL_CONSTANTS.C_MAX_SMOKE_SENSORS] OF INT;  (* Привязка дымовых датчиков к зонам эвакуации *)
  G_Evac_Leak_Zone_Map : ARRAY[1..GVL_CONSTANTS.C_MAX_FLOOD_SENSORS] OF INT;  (* Привязка датчиков протечки к зонам эвакуации *)
  G_Evac_Gas_Zone_Map : ARRAY[1..GVL_CONSTANTS.C_MAX_METHANE_SENSORS] OF INT;  (* Привязка газовых датчиков к зонам эвакуации *)
  G_Evac_Zone_Names : ARRAY[1..32] OF STRING(80);  (* Человекочитаемые имена зон (помещения/крыло/этаж/сторона) *)
END_VAR

{attribute 'qualified_only'}
VAR_GLOBAL  (* GVL_TRACE *)
  G_Trace_Index : INT := 0;
  G_Trace_Max : INT := 100;
  G_Trace_Time : ARRAY[1..100] OF UDINT;
  G_Trace_Code : ARRAY[1..100] OF INT;
END_VAR

{attribute 'qualified_only'}
VAR_GLOBAL  (* GVL_HEALTH_BRIDGE *)
  G_Smoke_Detected : BOOL;
  G_Gas_Detected : BOOL;
  G_Leak_Detected : BOOL;
  G_Leak_Warning_Level : BOOL;
  G_CO_Warning_Level : BOOL;
  G_CO_Alarm_Level : BOOL;
  G_Last_Fault_Event_Text : STRING(255);
END_VAR

{attribute 'qualified_only'}
VAR_GLOBAL  (* GVL_TEST_INJECTION *)
  G_Inject_Enable : BOOL := FALSE;
  G_Inject_Gas_Level : REAL := 0.0;
  G_Inject_Force_Gas_Alarm_Reset : BOOL := FALSE;
  G_Inject_Force_IO_Offline : BOOL := FALSE;
  G_Scenario_Enable : BOOL := FALSE;
  G_Scenario_Auto_Run : BOOL := FALSE;
  G_Scenario_Reset_Request : BOOL := FALSE;
  G_Scenario_Current : INT := 0;
  G_Scenario_Step : INT := 0;
  G_Scenario_Done : BOOL := FALSE;
  G_Scenario_Failed : BOOL := FALSE;
  G_Scenario_Last_Result_Code : UDINT := 0;
  G_Scenario_Status_Msg : STRING(200) := 'Scenario runner idle';
  G_Test_Step : INT := 0;
  G_Test_Timer_MS : UDINT := 0;
END_VAR

{attribute 'qualified_only'}
VAR_GLOBAL RETAIN  (* GVL_Retain *)
  G_Initialized : BOOL := FALSE;  (* Флаг инициализации retain-переменных *)
  G_NVRAM_Data : ARRAY[0..12799] OF BYTE;  (* 100 * 128 = 12800 байт *)
  G_BlackBox_Buffer : ARRAY[0..GVL_CONSTANTS.C_MAX_BLACKBOX_RECORDS-1] OF ST_BlackBox_Record;
  G_BlackBox_LastIndex : INT;
  G_BlackBox_Frozen : BOOL;
  G_Presence_History : ARRAY[0..GVL_CONSTANTS.C_MAX_PRESENCE_HISTORY-1] OF WORD;  (* 168 часов * 6 записей в час = 1008 записей (битовая маска 16 ламп) *)
  G_History_Buffer : ARRAY[1..GVL_CONSTANTS.C_MAX_HISTORY_RECORDS] OF ST_History_Record;
  G_History_Write_Idx : INT := 1;
  G_History_Total_Events : UDINT;
  G_Boiler_Accumulated_MS : ARRAY[1..GVL_CONSTANTS.C_MAX_BOILERS] OF UDINT;
  G_Boiler_Work_Seconds : ARRAY[1..GVL_CONSTANTS.C_MAX_BOILERS] OF UDINT;
  G_Valve_Test_Results : ARRAY[1..GVL_CONSTANTS.C_MAX_MANIFOLDS] OF BOOL;
  G_Access_Codes : ARRAY[1..GVL_CONSTANTS.C_MAX_ACCESS_CODES] OF DWORD := [16#9BE3E0A3, 16#4A89A12D, 16#F4DBDF21, 16#90F59C65, 16#0972D346, 0, 0, 0, 0, 0];
  G_RFID_Tags : ARRAY[1..GVL_CONSTANTS.C_MAX_ACCESS_CODES] OF STRING(20) := ['A1B2C3D4', 'E5F67890', '', '', '', '', '', '', '', ''];
END_VAR

FUNCTION_BLOCK FB_Security_System_Manager
  VAR_INPUT
    VI_System_Time_MS : UDINT;
    VI_IsActivePLC : BOOL;
    VI_Arm_Request : BOOL;
    VI_Disarm_Request : BOOL;
    VI_PIN_Code : STRING(4);
    VI_RFID_Tag : STRING(20);
    VI_2FA_Code : STRING(6);
    VI_Config : ST_Security_Global_Config;
    VI_Current_TOD : TOD;
  END_VAR
  VAR_OUTPUT
    VO_Armed : BOOL;
    VO_Alarm_Active : BOOL;
    VO_Siren_Active : BOOL;
    VO_Status_Msg : STRING(200);
    VO_Send_Code_Req : BOOL;
    VO_Code_To_Send : STRING(6);
  END_VAR
  VAR_IN_OUT
    VI_Motion_Sensors : ARRAY[1..16] OF BOOL;
    VI_Door_Sensors : ARRAY[1..GVL_CONSTANTS.C_MAX_DOOR_SENSORS] OF BOOL;
    VI_Window_Sensors : ARRAY[1..16] OF BOOL;
    VI_Bypass_Motion : ARRAY[1..16] OF BOOL;
    VI_Bypass_Doors : ARRAY[1..GVL_CONSTANTS.C_MAX_DOOR_SENSORS] OF BOOL;
    VI_Bypass_Windows : ARRAY[1..16] OF BOOL;
  END_VAR
  VAR
    L_i : INT;
    L_Any_Sensor_Active : BOOL;
    L_Arm_Delay_Timer : FB_System_Timer;
    L_Alarm_Delay_Timer : FB_System_Timer;
    L_Arming_In_Progress : BOOL;
    L_Valid_PIN : BOOL;
    fbAccessCode : FB_AccessCode_Manager;
    fbTwoFactor : FB_TwoFactor_Auth;
    L_2FA_Required : BOOL;
    L_Disarm_Pending : BOOL;
    L_Reset_2FA : BOOL;
    L_Auto_Arm_Trigger : BOOL;
    R_Trig_Auto_Arm : R_TRIG;
  END_VAR

            IF NOT VI_IsActivePLC THEN
    VO_Armed := FALSE;
    VO_Alarm_Active := FALSE;
    VO_Siren_Active := FALSE;
    VO_Send_Code_Req := FALSE;
    VO_Code_To_Send := '';
    VO_Status_Msg := 'Охрана: резервный ПЛК';
    L_Arming_In_Progress := FALSE;
    L_Disarm_Pending := FALSE;
    L_2FA_Required := FALSE;
    L_Reset_2FA := FALSE;
    RETURN;
END_IF;

// 1. Проверка PIN-кода или RFID-метки через менеджер кодов
fbAccessCode(
    VI_System_Time_MS := VI_System_Time_MS,
    VI_IsActivePLC := VI_IsActivePLC,
    VI_Code_To_Check := VI_PIN_Code,
    VI_RFID_To_Check := VI_RFID_Tag,
    VI_Access_Codes := GVL_RETAIN.G_Access_Codes,
    VI_RFID_Tags := GVL_RETAIN.G_RFID_Tags,
    VO_Code_Valid => L_Valid_PIN
);

// 2. Логика постановки на охрану (с задержкой на выход)
L_Auto_Arm_Trigger := FALSE;
IF VI_Config.auto_arm_enabled THEN
    IF VI_Current_TOD >= UDINT_TO_TOD(VI_Config.auto_arm_time_ms) THEN
        L_Auto_Arm_Trigger := TRUE;
    END_IF;
END_IF;
R_Trig_Auto_Arm(CLK := L_Auto_Arm_Trigger);

IF ((VI_Arm_Request AND L_Valid_PIN) OR R_Trig_Auto_Arm.Q) AND NOT VO_Armed AND NOT L_Arming_In_Progress THEN
    // Проверка, что все двери/окна закрыты перед постановкой (с учетом байпаса)
    L_Any_Sensor_Active := FALSE;
    FOR L_i := 1 TO GVL_CONSTANTS.C_MAX_DOOR_SENSORS DO IF VI_Door_Sensors[L_i] AND NOT VI_Bypass_Doors[L_i] THEN L_Any_Sensor_Active := TRUE; END_IF; END_FOR;
    FOR L_i := 1 TO 16 DO IF VI_Window_Sensors[L_i] AND NOT VI_Bypass_Windows[L_i] THEN L_Any_Sensor_Active := TRUE; END_IF; END_FOR;
    
    IF NOT L_Any_Sensor_Active THEN
        L_Arming_In_Progress := TRUE;
        VO_Status_Msg := 'Постановка на охрану. Покиньте помещение.';
    ELSE
        VO_Status_Msg := 'Ошибка постановки: Открыты двери или окна';
    END_IF;
END_IF;

L_Arm_Delay_Timer(IN := L_Arming_In_Progress, PT := TO_TIME(VI_Config.exit_delay_seconds * 1000), VI_System_Time_MS := VI_System_Time_MS);
IF L_Arm_Delay_Timer.Q THEN
    L_Arming_In_Progress := FALSE;
    VO_Armed := TRUE;
    VO_Status_Msg := 'Система под охраной';
END_IF;

// 3. Логика снятия с охраны с 2FA
IF VI_Disarm_Request AND L_Valid_PIN AND VO_Armed THEN
    IF VI_Config.enable_2fa THEN
        L_Disarm_Pending := TRUE;
        L_2FA_Required := TRUE;
        VO_Status_Msg := 'Ожидание 2FA для снятия с охраны';
    ELSE
        // Снятие без 2FA
        VO_Armed := FALSE;
        VO_Alarm_Active := FALSE;
        VO_Siren_Active := FALSE;
        L_Arming_In_Progress := FALSE;
        VO_Status_Msg := 'Система снята с охраны';
    END_IF;
END_IF;

fbTwoFactor(
    VI_System_Time_MS := VI_System_Time_MS,
    VI_Start_Auth := L_2FA_Required,
    VI_Method := E_TwoFactor_Method.TF_METHOD_TOTP, // Для примера
    VI_User_Code := VI_2FA_Code, // Используем отдельный вход для 2FA кода
    VI_Reset_Success := L_Reset_2FA
);

VO_Send_Code_Req := fbTwoFactor.VO_Send_Code_Req;
VO_Code_To_Send := fbTwoFactor.VO_Code_To_Send;

IF L_Disarm_Pending AND fbTwoFactor.VO_State.Is_Success THEN
    VO_Armed := FALSE;
    VO_Alarm_Active := FALSE;
    VO_Siren_Active := FALSE;
    L_Arming_In_Progress := FALSE;
    L_Disarm_Pending := FALSE;
    L_2FA_Required := FALSE;
    L_Reset_2FA := TRUE;
    VO_Status_Msg := 'Система снята с охраны';
ELSIF L_Disarm_Pending AND fbTwoFactor.VO_State.Is_Locked THEN
    L_Disarm_Pending := FALSE;
    L_2FA_Required := FALSE;
    L_Reset_2FA := FALSE;
    VO_Status_Msg := 'Ошибка 2FA: Превышено количество попыток';
ELSE
    L_Reset_2FA := FALSE;
END_IF;

// 4. Логика тревоги (с задержкой на вход)
IF VO_Armed THEN
    L_Any_Sensor_Active := FALSE;
    FOR L_i := 1 TO 16 DO IF VI_Motion_Sensors[L_i] AND NOT VI_Bypass_Motion[L_i] THEN L_Any_Sensor_Active := TRUE; END_IF; END_FOR;
    FOR L_i := 1 TO GVL_CONSTANTS.C_MAX_DOOR_SENSORS DO IF VI_Door_Sensors[L_i] AND NOT VI_Bypass_Doors[L_i] THEN L_Any_Sensor_Active := TRUE; END_IF; END_FOR;
    FOR L_i := 1 TO 16 DO IF VI_Window_Sensors[L_i] AND NOT VI_Bypass_Windows[L_i] THEN L_Any_Sensor_Active := TRUE; END_IF; END_FOR;
    
    // Защелкиваем факт нарушения периметра, чтобы кратковременное срабатывание датчика не сбрасывало таймер
    IF L_Any_Sensor_Active THEN
        L_Alarm_Delay_Timer.IN := TRUE;
    END_IF;
    
    L_Alarm_Delay_Timer(PT := TO_TIME(VI_Config.entry_delay_seconds * 1000), VI_System_Time_MS := VI_System_Time_MS);
    
    IF L_Alarm_Delay_Timer.Q THEN
        VO_Alarm_Active := TRUE;
        VO_Siren_Active := TRUE;
        VO_Status_Msg := 'ТРЕВОГА! Нарушение периметра';
    ELSIF L_Alarm_Delay_Timer.IN THEN
        VO_Status_Msg := 'Внимание! Введите PIN-код для отмены тревоги';
    END_IF;
ELSE
    L_Alarm_Delay_Timer(IN := FALSE, PT := T#0s, VI_System_Time_MS := VI_System_Time_MS); // Сброс таймера при снятии с охраны
END_IF;
// >>> BULK_SYNC_ANCHOR: FB_Security_System_Manager <<<
          
END_FUNCTION_BLOCK

FUNCTION_BLOCK FB_System_Timebase
  VAR
    L_Time_Diff : UDINT;
  END_VAR

            // ==============================================================================
// System timebase helper
//
// Internal helper for PRG_System.
// Owns PLC runtime clock projection into GVL_STATUS:
// - monotonic system milliseconds
// - time-of-day milliseconds
// - day of week / day of year rollover
// - TOD representation
// ==============================================================================



GVL_STATUS.G_System_Time_MS := TIME_TO_UDINT(TIME());

L_Time_Diff := SEL(
    GVL_STATUS.G_System_Time_MS >= GVL_STATUS.G_Last_System_Time_MS,
    GVL_STATUS.G_System_Time_MS - GVL_STATUS.G_Last_System_Time_MS,
    (4294967295 - GVL_STATUS.G_Last_System_Time_MS) + GVL_STATUS.G_System_Time_MS + 1
);

GVL_STATUS.G_Time_Of_Day_MS := (GVL_STATUS.G_Time_Of_Day_MS + L_Time_Diff) MOD 86400000;

IF GVL_STATUS.G_Time_Of_Day_MS < L_Time_Diff THEN
    GVL_STATUS.G_Current_Day := (GVL_STATUS.G_Current_Day MOD 7) + 1;
    GVL_STATUS.G_Day_Of_Year := (GVL_STATUS.G_Day_Of_Year MOD 365) + 1;
END_IF;

GVL_STATUS.G_Last_System_Time_MS := GVL_STATUS.G_System_Time_MS;
GVL_STATUS.G_Current_TOD := UDINT_TO_TOD(GVL_STATUS.G_Time_Of_Day_MS);

// >>> BULK_SYNC_ANCHOR: FB_System_Timebase <<<
          
END_FUNCTION_BLOCK

FUNCTION_BLOCK FB_Trace_Logger
  VAR_INPUT
    VI_Event_Code : INT;
    VI_System_Time : UDINT;
  END_VAR

            GVL_TRACE.G_Trace_Index := GVL_TRACE.G_Trace_Index + 1;
IF GVL_TRACE.G_Trace_Index > GVL_TRACE.G_Trace_Max THEN
    GVL_TRACE.G_Trace_Index := 1;
END_IF;

GVL_TRACE.G_Trace_Time[GVL_TRACE.G_Trace_Index] := VI_System_Time;
GVL_TRACE.G_Trace_Code[GVL_TRACE.G_Trace_Index] := VI_Event_Code;
          
END_FUNCTION_BLOCK

FUNCTION_BLOCK FB_Command_Deduplication
  VAR_INPUT
    VI_Command_ID : UDINT;
    VI_Command_Type : E_Gateway_Command_Type;
    VI_Command_Value : REAL;
    VI_System_Time_MS : UDINT;
  END_VAR
  VAR_OUTPUT
    VO_Is_New_Command : BOOL;
    VO_Processed_ID : UDINT;
  END_VAR
  VAR
    L_Processed_History : ARRAY[0..GVL_CONSTANTS.C_MAX_DEDUPLICATION_HISTORY-1] OF UDINT;
    L_Processed_Times : ARRAY[0..GVL_CONSTANTS.C_MAX_DEDUPLICATION_HISTORY-1] OF UDINT;
    L_History_Index : INT := 0;
    L_i : INT;
    L_Found : BOOL;
  END_VAR

            // Check if command ID is already in history
L_Found := FALSE;
FOR L_i := 0 TO GVL_CONSTANTS.C_MAX_DEDUPLICATION_HISTORY-1 DO
    IF L_Processed_History[L_i] = VI_Command_ID AND VI_Command_ID <> 0 THEN
        // Check if the command is not too old (e.g., 1 hour = 3600000 ms)
        IF (VI_System_Time_MS - L_Processed_Times[L_i]) < 3600000 THEN
            L_Found := TRUE;
            EXIT;
        END_IF;
    END_IF;
END_FOR;

IF NOT L_Found AND VI_Command_ID <> 0 THEN
    // New command detected
    VO_Is_New_Command := TRUE;
    VO_Processed_ID := VI_Command_ID;
    
    // Add to history
    L_Processed_History[L_History_Index] := VI_Command_ID;
    L_Processed_Times[L_History_Index] := VI_System_Time_MS;
    L_History_Index := L_History_Index + 1;
    IF L_History_Index > GVL_CONSTANTS.C_MAX_DEDUPLICATION_HISTORY-1 THEN
        L_History_Index := 0;
    END_IF;
ELSE
    // Duplicate or empty command
    VO_Is_New_Command := FALSE;
    VO_Processed_ID := 0;
END_IF;
          
END_FUNCTION_BLOCK

FUNCTION_BLOCK FB_Sensor_Calibration
  VAR_INPUT
    VI_Sensor_ID : UDINT;
    VI_Reference_Value : REAL;
    VI_Current_Value : REAL;
    VI_Apply : BOOL;
  END_VAR
  VAR_OUTPUT
    VO_Offset : REAL;
    VO_Multiplier : REAL := 1.0;
    VO_Done : BOOL;
  END_VAR
  VAR
    L_Applied : BOOL;
  END_VAR

            IF VI_Apply AND NOT L_Applied THEN
    // Простая калибровка смещением (одноточечная)
    VO_Offset := VI_Reference_Value - VI_Current_Value;
    VO_Done := TRUE;
    L_Applied := TRUE;
ELSIF NOT VI_Apply THEN
    VO_Done := FALSE;
    L_Applied := FALSE;
END_IF;
          
END_FUNCTION_BLOCK

FUNCTION_BLOCK FB_System_Persist_Manager
  VAR_INPUT
    VI_System_Time_MS : UDINT;
    VI_IsActivePLC : BOOL;
  END_VAR
  VAR_IN_OUT
    VIO_Persist_Buffer : ARRAY[0..4] OF BYTE;
    VIO_Last_Written_Persist_Buffer : ARRAY[0..4] OF BYTE;
    VIO_Persist_Buffer_Changed : BOOL;
    VIO_Last_Persist_Write_MS : UDINT;
    VIO_NVRAM_Cmd : BYTE;
    VIO_NVRAM_Offset : UDINT;
    VIO_NVRAM_Done : BOOL;
    VIO_NVRAM_Err : BOOL;
    VIO_NVRAM_ErrID : UDINT;
  END_VAR
  VAR
    fbNVRAMManager : FB_NVRAM_Manager;
  END_VAR

            // ==============================================================================
// System persist manager helper
//
// Internal helper for PRG_System.
// Owns persistent snapshot packing, controlled NVRAM write gating,
// FB_NVRAM_Manager call, and last-written buffer tracking.
// ==============================================================================



// Pack persistent snapshot into compact byte buffer for controlled NVRAM mirroring
VIO_Persist_Buffer[0] := TO_BYTE(TO_INT(GVL_STATE.G_System_Mode));
IF GVL_PERSISTENT.P_Safety_Gas_Latched THEN
    VIO_Persist_Buffer[1] := BYTE#1;
ELSE
    VIO_Persist_Buffer[1] := BYTE#0;
END_IF;
IF GVL_PERSISTENT.P_Safety_Smoke_Latched THEN
    VIO_Persist_Buffer[2] := BYTE#1;
ELSE
    VIO_Persist_Buffer[2] := BYTE#0;
END_IF;
IF GVL_PERSISTENT.P_Safety_Leak_Latched THEN
    VIO_Persist_Buffer[3] := BYTE#1;
ELSE
    VIO_Persist_Buffer[3] := BYTE#0;
END_IF;
IF GVL_PERSISTENT.P_DHW_Heating_Active THEN
    VIO_Persist_Buffer[4] := BYTE#1;
ELSE
    VIO_Persist_Buffer[4] := BYTE#0;
END_IF;

VIO_Persist_Buffer_Changed :=
    (VIO_Persist_Buffer[0] <> VIO_Last_Written_Persist_Buffer[0]) OR
    (VIO_Persist_Buffer[1] <> VIO_Last_Written_Persist_Buffer[1]) OR
    (VIO_Persist_Buffer[2] <> VIO_Last_Written_Persist_Buffer[2]) OR
    (VIO_Persist_Buffer[3] <> VIO_Last_Written_Persist_Buffer[3]) OR
    (VIO_Persist_Buffer[4] <> VIO_Last_Written_Persist_Buffer[4]);

VIO_NVRAM_Cmd := 0;
VIO_NVRAM_Offset := 0;

IF GVL_CONFIG.G_HMI_Apply_Settings THEN
    // explicit config apply may request a controlled write
    VIO_NVRAM_Cmd := 1;
    GVL_CONFIG.G_HMI_Apply_Settings := FALSE;

ELSIF VIO_Persist_Buffer_Changed THEN
    // controlled write: no more often than once per 60 seconds
    IF (VIO_Last_Persist_Write_MS = 0) OR
       ((VI_System_Time_MS - VIO_Last_Persist_Write_MS) >= 60000) THEN
        VIO_NVRAM_Cmd := 1;
    END_IF;
END_IF;

fbNVRAMManager(
    VI_Command := VIO_NVRAM_Cmd,
    VI_Offset := VIO_NVRAM_Offset,
    VI_DataRef := VIO_Persist_Buffer[0],
    VI_DataSize := 5,
    VI_System_Time_MS := VI_System_Time_MS,
    VI_Operator_ID := 'SYSTEM',
    VI_IsActivePLC := VI_IsActivePLC,
    VI_TwoPersonConfirmation := FALSE,
    VO_Done => VIO_NVRAM_Done,
    VO_Error => VIO_NVRAM_Err,
    VO_ErrorID => VIO_NVRAM_ErrID
);

IF (VIO_NVRAM_Cmd = 1) AND VIO_NVRAM_Done AND NOT VIO_NVRAM_Err THEN
    VIO_Last_Written_Persist_Buffer[0] := VIO_Persist_Buffer[0];
    VIO_Last_Written_Persist_Buffer[1] := VIO_Persist_Buffer[1];
    VIO_Last_Written_Persist_Buffer[2] := VIO_Persist_Buffer[2];
    VIO_Last_Written_Persist_Buffer[3] := VIO_Persist_Buffer[3];
    VIO_Last_Written_Persist_Buffer[4] := VIO_Persist_Buffer[4];
    VIO_Last_Persist_Write_MS := VI_System_Time_MS;
END_IF;

// >>> BULK_SYNC_ANCHOR: FB_System_Persist_Manager <<<
          
END_FUNCTION_BLOCK

FUNCTION_BLOCK FB_Lighting_Blinds_Manager
  VAR_INPUT
    VI_System_Time_MS : UDINT;
    VI_IsActivePLC : BOOL;
    VI_Current_Scenario : E_SCENARIO_TYPE;
    VI_Away_Level : BYTE;
    VI_Simulation_Active : BOOL;
    VI_Is_Night : BOOL;
    VI_System_Mode : E_System_Operating_Mode;
  END_VAR
  VAR_OUTPUT
    VO_Lighting_Levels : ARRAY[1..32] OF BYTE;
    VO_Blinds_Positions : ARRAY[1..GVL_CONSTANTS.C_MAX_BLINDS] OF BYTE;
    VO_Wet_Zone_Light_Active : ARRAY[1..GVL_CONSTANTS.C_MAX_WET_ZONES] OF BOOL;
  END_VAR
  VAR_IN_OUT
    VI_Manual_Light_Override : ARRAY[1..32] OF BYTE;
    VI_Manual_Blinds_Override : ARRAY[1..GVL_CONSTANTS.C_MAX_BLINDS] OF BYTE;
    VI_Simulation_Lights : ARRAY[1..32] OF BOOL;
    VI_Physical_Switches : ARRAY[1..32] OF BOOL;
    VI_Motion_Sensors : ARRAY[1..32] OF BOOL;
    VI_Rule_Actions : ARRAY[1..GVL_CONSTANTS.C_MAX_RULES] OF ST_Rule_Action;
    VI_IO_Modules_Online : ARRAY[1..GVL_CONSTANTS.C_MAX_MODULES] OF BOOL;
    VI_Wet_Zone_Map : ARRAY[1..32] OF BOOL;
    VI_Scenario_Configs : ARRAY[1..GVL_CONSTANTS.C_MAX_SCENARIOS] OF ST_Scenario_Config;
  END_VAR
  VAR
    L_i : INT;
    L_j : INT;
    L_Base_Light : BYTE;
    L_Base_Blinds : BYTE;
    L_Target_Base_Light : BYTE;
    L_Target_Base_Blinds : BYTE;
    L_Prev_Scenario : E_SCENARIO_TYPE;
    L_Transition_Light : FB_Scenario_Transition_Controller;
    L_Transition_Blinds : FB_Scenario_Transition_Controller;
    L_Light_States : ARRAY[1..32] OF BOOL;
    L_Prev_Switches : ARRAY[1..32] OF BOOL;
    L_Prev_Motion_Q : ARRAY[1..32] OF BOOL;
    L_Manual_Override : ARRAY[1..32] OF BOOL;
    L_Motion_Timers : ARRAY[1..32] OF FB_System_Timer_TOF;
    L_Rule_Light_Active : BOOL;
    L_Rule_Light_Val : BYTE;
    L_Rule_Blinds_Active : BOOL;
    L_Rule_Blinds_Val : BYTE;
    L_Wet_Zone_Idx : INT;
    L_Effective_Scenario : E_SCENARIO_TYPE;
    L_Effective_Simulation_Active : BOOL;
  END_VAR

            // Менеджер управления освещением и шторами/жалюзи.
// Обеспечивает работу по сценариями, датчикам движения, физическим выключателям и правилам.


IF NOT VI_IsActivePLC THEN RETURN; END_IF;


GVL_STATE.G_Lighting_IO_Fault := FALSE;
GVL_STATE.G_Lighting_Subsystem_Degraded := FALSE;

L_Effective_Scenario := VI_Current_Scenario;
L_Effective_Simulation_Active := VI_Simulation_Active;

CASE VI_System_Mode OF
    E_System_Operating_Mode.MODE_SAFE_STOP:
        FOR L_j := 1 TO 32 DO
            VO_Lighting_Levels[L_j] := 0;
        END_FOR;
        FOR L_j := 1 TO GVL_CONSTANTS.C_MAX_BLINDS DO
            VO_Blinds_Positions[L_j] := 100;
        END_FOR;
        FOR L_j := 1 TO GVL_CONSTANTS.C_MAX_WET_ZONES DO
            VO_Wet_Zone_Light_Active[L_j] := FALSE;
        END_FOR;
        RETURN;
    E_System_Operating_Mode.MODE_FREEZE_PROTECTION:
        L_Effective_Scenario := E_SCENARIO_TYPE.SCENARIO_NONE;
        L_Effective_Simulation_Active := FALSE;
    E_System_Operating_Mode.MODE_DEGRADED:
        L_Effective_Simulation_Active := FALSE;
END_CASE;

// Инициализация индекса мокрых зон
L_Wet_Zone_Idx := 1;
// Сброс массива мокрых зон
FOR L_i := 1 TO GVL_CONSTANTS.C_MAX_WET_ZONES DO
    VO_Wet_Zone_Light_Active[L_i] := FALSE;
END_FOR;

// Проверка связи с модулями ввода-вывода
FOR L_i := 1 TO GVL_CONSTANTS.C_MAX_MODULES DO
    IF NOT VI_IO_Modules_Online[L_i] THEN
        GVL_STATE.G_Lighting_IO_Fault := TRUE;
GVL_STATE.G_Lighting_Subsystem_Degraded := TRUE;
        // Переход в безопасное состояние при потере связи (свет выкл, шторы открыты для эвакуации)
        FOR L_j := 1 TO 32 DO
            VO_Lighting_Levels[L_j] := 0;
        END_FOR;
        FOR L_j := 1 TO GVL_CONSTANTS.C_MAX_BLINDS DO
            VO_Blinds_Positions[L_j] := 100;
        END_FOR;
        RETURN;
    END_IF;
END_FOR;

// 1. Определение целевых уровней по сценарию (ТЗ 7.1)
IF L_Effective_Scenario >= 1 AND L_Effective_Scenario <= GVL_CONSTANTS.C_MAX_SCENARIOS THEN
    L_Target_Base_Light := VI_Scenario_Configs[L_Effective_Scenario].lighting_level_base;
    L_Target_Base_Blinds := VI_Scenario_Configs[L_Effective_Scenario].blinds_position_percent;
ELSE
    L_Target_Base_Light := 100;
    L_Target_Base_Blinds := 100;
END_IF;

// Корректировка по астрономическому таймеру
IF VI_Is_Night AND L_Effective_Scenario <> E_SCENARIO_TYPE.SCENARIO_AWAY AND L_Effective_Scenario <> E_SCENARIO_TYPE.SCENARIO_SLEEP THEN
    L_Target_Base_Blinds := 0; // Закрывать шторы ночью
END_IF;

// Плавный переход при смене сценария
IF L_Effective_Scenario <> L_Prev_Scenario THEN
    L_Transition_Light(
        VI_System_Time := VI_System_Time_MS,
        VI_Start_Time := VI_System_Time_MS,
        VI_Duration := 5000, // 5 секунд на плавное изменение света
        VI_Start_Value := TO_REAL(L_Base_Light),
        VI_End_Value := TO_REAL(L_Target_Base_Light)
    );
    L_Transition_Blinds(
        VI_System_Time := VI_System_Time_MS,
        VI_Start_Time := VI_System_Time_MS,
        VI_Duration := 10000, // 10 секунд на плавное изменение штор
        VI_Start_Value := TO_REAL(L_Base_Blinds),
        VI_End_Value := TO_REAL(L_Target_Base_Blinds)
    );
    L_Prev_Scenario := L_Effective_Scenario;
ELSE
    L_Transition_Light(
        VI_System_Time := VI_System_Time_MS,
        VI_Start_Time := L_Transition_Light.VI_Start_Time,
        VI_Duration := L_Transition_Light.VI_Duration,
        VI_Start_Value := L_Transition_Light.VI_Start_Value,
        VI_End_Value := TO_REAL(L_Target_Base_Light)
    );
    L_Transition_Blinds(
        VI_System_Time := VI_System_Time_MS,
        VI_Start_Time := L_Transition_Blinds.VI_Start_Time,
        VI_Duration := L_Transition_Blinds.VI_Duration,
        VI_Start_Value := L_Transition_Blinds.VI_Start_Value,
        VI_End_Value := TO_REAL(L_Target_Base_Blinds)
    );
END_IF;

L_Base_Light := TO_BYTE(L_Transition_Light.VO_Current_Value);
L_Base_Blinds := TO_BYTE(L_Transition_Blinds.VO_Current_Value);

// 2. Управление освещением
FOR L_i := 1 TO 32 DO
    L_Rule_Light_Active := FALSE;
    L_Rule_Light_Val := 0;
    
    // Проверка правил
    FOR L_j := 1 TO GVL_CONSTANTS.C_MAX_RULES DO
        IF VI_Rule_Actions[L_j].Active AND VI_Rule_Actions[L_j].Target_ID = L_i THEN
            IF VI_Rule_Actions[L_j].Action_Type = E_Rule_Action_Type.ACTION_SET_LIGHTING_BASE THEN
                L_Rule_Light_Active := TRUE;
                L_Rule_Light_Val := REAL_TO_BYTE(VI_Rule_Actions[L_j].Value);
                L_Light_States[L_i] := (L_Rule_Light_Val > 0);
            ELSIF VI_Rule_Actions[L_j].Action_Type = E_Rule_Action_Type.ACTION_TOGGLE_LIGHTING AND VI_Rule_Actions[L_j].Triggered THEN
                L_Light_States[L_i] := NOT L_Light_States[L_i];
            END_IF;
        END_IF;
    END_FOR;

    // Приоритет 1: Физические выключатели (ТЗ 1.0)
    IF VI_Physical_Switches[L_i] AND NOT L_Prev_Switches[L_i] THEN
        L_Light_States[L_i] := NOT L_Light_States[L_i];
        L_Manual_Override[L_i] := TRUE; // Запоминаем ручное переопределение
    END_IF;
    L_Prev_Switches[L_i] := VI_Physical_Switches[L_i];

    // Приоритет 2: Датчики движения (ТЗ 2.0)
    // Защита от дребезга и удержание сигнала движения с помощью TOF
    L_Motion_Timers[L_i](IN := VI_Motion_Sensors[L_i], PT := T#5m, VI_System_Time_MS := VI_System_Time_MS);
    
    // Сброс ручного переопределения, когда комната становится пустой (задний фронт таймера движения)
    IF L_Prev_Motion_Q[L_i] AND NOT L_Motion_Timers[L_i].Q THEN
        L_Manual_Override[L_i] := FALSE;
    END_IF;
    L_Prev_Motion_Q[L_i] := L_Motion_Timers[L_i].Q;

    IF L_Motion_Timers[L_i].Q THEN
        IF NOT L_Manual_Override[L_i] THEN
            L_Light_States[L_i] := TRUE;
        END_IF;
    ELSE
        // Выключаем свет только если нет ручного переопределения
        IF NOT L_Manual_Override[L_i] THEN
            L_Light_States[L_i] := FALSE;
        END_IF;
    END_IF;

    // Приоритет 3: Симуляция (только в режиме Away)
    IF L_Effective_Scenario = E_SCENARIO_TYPE.SCENARIO_AWAY AND L_Effective_Simulation_Active THEN
        L_Light_States[L_i] := VI_Simulation_Lights[L_i];
    END_IF;

    // Приоритет 4: Ручное управление и правила
    IF VI_Manual_Light_Override[L_i] > 0 THEN
        VO_Lighting_Levels[L_i] := VI_Manual_Light_Override[L_i];
    ELSIF L_Rule_Light_Active THEN
        VO_Lighting_Levels[L_i] := L_Rule_Light_Val;
    ELSE
        VO_Lighting_Levels[L_i] := SEL(L_Light_States[L_i], 0, L_Base_Light);
    END_IF;
    
    // 5. Мокрые зоны
    IF VI_Wet_Zone_Map[L_i] AND L_Wet_Zone_Idx <= GVL_CONSTANTS.C_MAX_WET_ZONES THEN
        VO_Wet_Zone_Light_Active[L_Wet_Zone_Idx] := (VO_Lighting_Levels[L_i] > 10);
        L_Wet_Zone_Idx := L_Wet_Zone_Idx + 1;
    END_IF;
END_FOR;

// 3. Управление шторами
FOR L_i := 1 TO GVL_CONSTANTS.C_MAX_BLINDS DO
    L_Rule_Blinds_Active := FALSE;
    L_Rule_Blinds_Val := 0;
    
    // Проверка правил
    FOR L_j := 1 TO GVL_CONSTANTS.C_MAX_RULES DO
        IF VI_Rule_Actions[L_j].Active AND VI_Rule_Actions[L_j].Target_ID = L_i THEN
            IF VI_Rule_Actions[L_j].Action_Type = E_Rule_Action_Type.ACTION_SET_BLINDS THEN
                L_Rule_Blinds_Active := TRUE;
                L_Rule_Blinds_Val := REAL_TO_BYTE(VI_Rule_Actions[L_j].Value);
            END_IF;
        END_IF;
    END_FOR;

    // Приоритет 1: Ручное управление
    IF VI_Manual_Blinds_Override[L_i] > 0 THEN
        VO_Blinds_Positions[L_i] := VI_Manual_Blinds_Override[L_i];
    // Приоритет 2: Правила
    ELSIF L_Rule_Blinds_Active THEN
        VO_Blinds_Positions[L_i] := L_Rule_Blinds_Val;
    // Приоритет 3: Сценарий
    ELSE
        VO_Blinds_Positions[L_i] := L_Base_Blinds;
    END_IF;
END_FOR;

// >>> BULK_SYNC_ANCHOR: FB_Lighting_Blinds_Manager <<<
          
END_FUNCTION_BLOCK

FUNCTION_BLOCK FB_Test_Result_Handler
  VAR_INPUT
    VI_Test_Passed : BOOL;
  END_VAR
  VAR
    L_Latched_Failure : BOOL;
  END_VAR

            // latch failure
IF NOT VI_Test_Passed THEN
    L_Latched_Failure := TRUE;
END_IF;

// enforce safe stop if failure latched
IF L_Latched_Failure THEN
    GVL_COMMAND.G_Gas_Valve_Close := TRUE;
    GVL_COMMAND.G_Close_Valve_35 := TRUE;
    GVL_COMMAND.G_Close_Valve_36 := TRUE;
END_IF;
          
END_FUNCTION_BLOCK

FUNCTION_BLOCK FB_Safety_Workflow_Manager
  VAR_INPUT
    VI_System_Time_MS : UDINT;
    VI_Water_Selective_Recover : BOOL;
    VI_Gas_Selective_Recover : BOOL;
    VI_Water_Valve_Test_Open : BOOL;
    VI_Water_Valve_Test_Close : BOOL;
    VI_Water_Valve_Test_Confirm : BOOL;
    VI_Gas_Valve_Test_Open : BOOL;
    VI_Gas_Valve_Test_Close : BOOL;
    VI_Gas_Valve_Test_Confirm : BOOL;
  END_VAR
  VAR_OUTPUT
    VO_Water_Selective_Recover_Edge : BOOL;
    VO_Gas_Selective_Recover_Edge : BOOL;
    VO_Water_Valve_Test_Open_Edge : BOOL;
    VO_Water_Valve_Test_Close_Edge : BOOL;
    VO_Water_Valve_Test_Confirm_Edge : BOOL;
    VO_Gas_Valve_Test_Open_Edge : BOOL;
    VO_Gas_Valve_Test_Close_Edge : BOOL;
    VO_Gas_Valve_Test_Confirm_Edge : BOOL;
    VO_Water_Test_Active : BOOL;
    VO_Gas_Test_Active : BOOL;
    VO_Water_Test_Timeout_Close_Required : BOOL;
    VO_Gas_Test_Timeout_Close_Required : BOOL;
  END_VAR
  VAR
    L_CMD_Water_Selective_Recover_Prev : BOOL;
    L_CMD_Gas_Selective_Recover_Prev : BOOL;
    L_CMD_Water_Valve_Test_Open_Prev : BOOL;
    L_CMD_Water_Valve_Test_Close_Prev : BOOL;
    L_CMD_Water_Valve_Test_Confirm_Prev : BOOL;
    L_CMD_Gas_Valve_Test_Open_Prev : BOOL;
    L_CMD_Gas_Valve_Test_Close_Prev : BOOL;
    L_CMD_Gas_Valve_Test_Confirm_Prev : BOOL;
    L_Water_Test_Active : BOOL;
    L_Water_Test_Deadline : UDINT;
    L_Gas_Test_Active : BOOL;
    L_Gas_Test_Deadline : UDINT;
  END_VAR

            VO_Water_Test_Timeout_Close_Required := FALSE;
VO_Gas_Test_Timeout_Close_Required := FALSE;

VO_Water_Selective_Recover_Edge := VI_Water_Selective_Recover AND NOT L_CMD_Water_Selective_Recover_Prev;
VO_Gas_Selective_Recover_Edge := VI_Gas_Selective_Recover AND NOT L_CMD_Gas_Selective_Recover_Prev;
VO_Water_Valve_Test_Open_Edge := VI_Water_Valve_Test_Open AND NOT L_CMD_Water_Valve_Test_Open_Prev;
VO_Water_Valve_Test_Close_Edge := VI_Water_Valve_Test_Close AND NOT L_CMD_Water_Valve_Test_Close_Prev;
VO_Water_Valve_Test_Confirm_Edge := VI_Water_Valve_Test_Confirm AND NOT L_CMD_Water_Valve_Test_Confirm_Prev;
VO_Gas_Valve_Test_Open_Edge := VI_Gas_Valve_Test_Open AND NOT L_CMD_Gas_Valve_Test_Open_Prev;
VO_Gas_Valve_Test_Close_Edge := VI_Gas_Valve_Test_Close AND NOT L_CMD_Gas_Valve_Test_Close_Prev;
VO_Gas_Valve_Test_Confirm_Edge := VI_Gas_Valve_Test_Confirm AND NOT L_CMD_Gas_Valve_Test_Confirm_Prev;

L_CMD_Water_Selective_Recover_Prev := VI_Water_Selective_Recover;
L_CMD_Gas_Selective_Recover_Prev := VI_Gas_Selective_Recover;
L_CMD_Water_Valve_Test_Open_Prev := VI_Water_Valve_Test_Open;
L_CMD_Water_Valve_Test_Close_Prev := VI_Water_Valve_Test_Close;
L_CMD_Water_Valve_Test_Confirm_Prev := VI_Water_Valve_Test_Confirm;
L_CMD_Gas_Valve_Test_Open_Prev := VI_Gas_Valve_Test_Open;
L_CMD_Gas_Valve_Test_Close_Prev := VI_Gas_Valve_Test_Close;
L_CMD_Gas_Valve_Test_Confirm_Prev := VI_Gas_Valve_Test_Confirm;

IF VO_Water_Valve_Test_Open_Edge THEN
    L_Water_Test_Active := TRUE;
    L_Water_Test_Deadline := VI_System_Time_MS + 60000;
END_IF;

IF L_Water_Test_Active THEN
    IF VI_System_Time_MS >= L_Water_Test_Deadline THEN
        L_Water_Test_Active := FALSE;
        VO_Water_Test_Timeout_Close_Required := TRUE;
    END_IF;
END_IF;

IF VO_Gas_Valve_Test_Open_Edge THEN
    L_Gas_Test_Active := TRUE;
    L_Gas_Test_Deadline := VI_System_Time_MS + 60000;
END_IF;

IF L_Gas_Test_Active THEN
    IF VI_System_Time_MS >= L_Gas_Test_Deadline THEN
        L_Gas_Test_Active := FALSE;
        VO_Gas_Test_Timeout_Close_Required := TRUE;
    END_IF;
END_IF;

VO_Water_Test_Active := L_Water_Test_Active;
VO_Gas_Test_Active := L_Gas_Test_Active;
          
END_FUNCTION_BLOCK

FUNCTION_BLOCK FB_HMAC_SHA1
  VAR_INPUT
    KeyLength : INT;
    MessageLength : INT;
  END_VAR
  VAR_OUTPUT
    Hash : ARRAY[0..19] OF BYTE;
    Done : BOOL;
  END_VAR
  VAR_IN_OUT
    Key : ARRAY[0..63] OF BYTE;
    Message : ARRAY[0..7] OF BYTE;
  END_VAR
  VAR
    i : INT;
    K_ipad : ARRAY[0..63] OF BYTE;
    K_opad : ARRAY[0..63] OF BYTE;
    InnerData : ARRAY[0..127] OF BYTE;
    OuterData : ARRAY[0..127] OF BYTE;
    InnerHash : ARRAY[0..19] OF BYTE;
    FB_SHA1_Inner : FB_SHA1;
    FB_SHA1_Outer : FB_SHA1;
  END_VAR

            // 1. Prepare K_ipad and K_opad
FOR i := 0 TO 63 DO
    IF i < KeyLength THEN
        K_ipad[i] := Key[i] XOR 16#36;
        K_opad[i] := Key[i] XOR 16#5C;
    ELSE
        K_ipad[i] := 16#36;
        K_opad[i] := 16#5C;
    END_IF;
END_FOR;

// 2. Inner Hash: SHA1(K_ipad || Message)
FOR i := 0 TO 63 DO
    InnerData[i] := K_ipad[i];
END_FOR;
FOR i := 0 TO MessageLength - 1 DO
    InnerData[64 + i] := Message[i];
END_FOR;

FB_SHA1_Inner(Data := InnerData, Length := 64 + MessageLength, Hash => InnerHash);

// 3. Outer Hash: SHA1(K_opad || InnerHash)
FOR i := 0 TO 63 DO
    OuterData[i] := K_opad[i];
END_FOR;
FOR i := 0 TO 19 DO
    OuterData[64 + i] := InnerHash[i];
END_FOR;

FB_SHA1_Outer(Data := OuterData, Length := 84, Hash => Hash);

Done := TRUE;
          
END_FUNCTION_BLOCK

FUNCTION_BLOCK FB_Maintenance_Access
  VAR_INPUT
    VI_System_Time : UDINT;
    VI_Activate : BOOL;
    VI_Duration : UDINT := 60;
  END_VAR
  VAR_OUTPUT
    VO_Active : BOOL;
    VO_Time_Left : UDINT;
  END_VAR
  VAR
    L_Start_Time : UDINT;
    L_elapsed : UDINT;
  END_VAR

            IF VI_Activate AND NOT VO_Active THEN
    VO_Active := TRUE;
    L_Start_Time := VI_System_Time;
END_IF;

IF VO_Active THEN
    L_elapsed := (SEL(VI_System_Time >= L_Start_Time, VI_System_Time - L_Start_Time, (4294967295 - L_Start_Time) + VI_System_Time + 1)) / GVL_CONSTANTS.C_MS_IN_MINUTE;
    IF L_elapsed >= VI_Duration THEN
        VO_Active := FALSE;
        VO_Time_Left := 0;
    ELSE
        VO_Time_Left := VI_Duration - L_elapsed;
    END_IF;
ELSE
    VO_Time_Left := 0;
END_IF;
          
END_FUNCTION_BLOCK

FUNCTION_BLOCK FB_Sensor_Calibration_Processor
  VAR_INPUT
    VI_Raw_Value : REAL;
    VI_Record : ST_Sensor_Calibration_Record;
  END_VAR
  VAR_OUTPUT
    VO_Calibrated_Value : REAL;
  END_VAR

            VO_Calibrated_Value := (VI_Raw_Value * VI_Record.multiplier) + VI_Record.offset;
          
END_FUNCTION_BLOCK

FUNCTION_BLOCK FB_LogEvent
  VAR_INPUT
    VI_Event_Type : UINT;
    VI_Timestamp : UDINT;
    VI_Param1 : UDINT;
    VI_Param2 : UDINT;
  END_VAR

